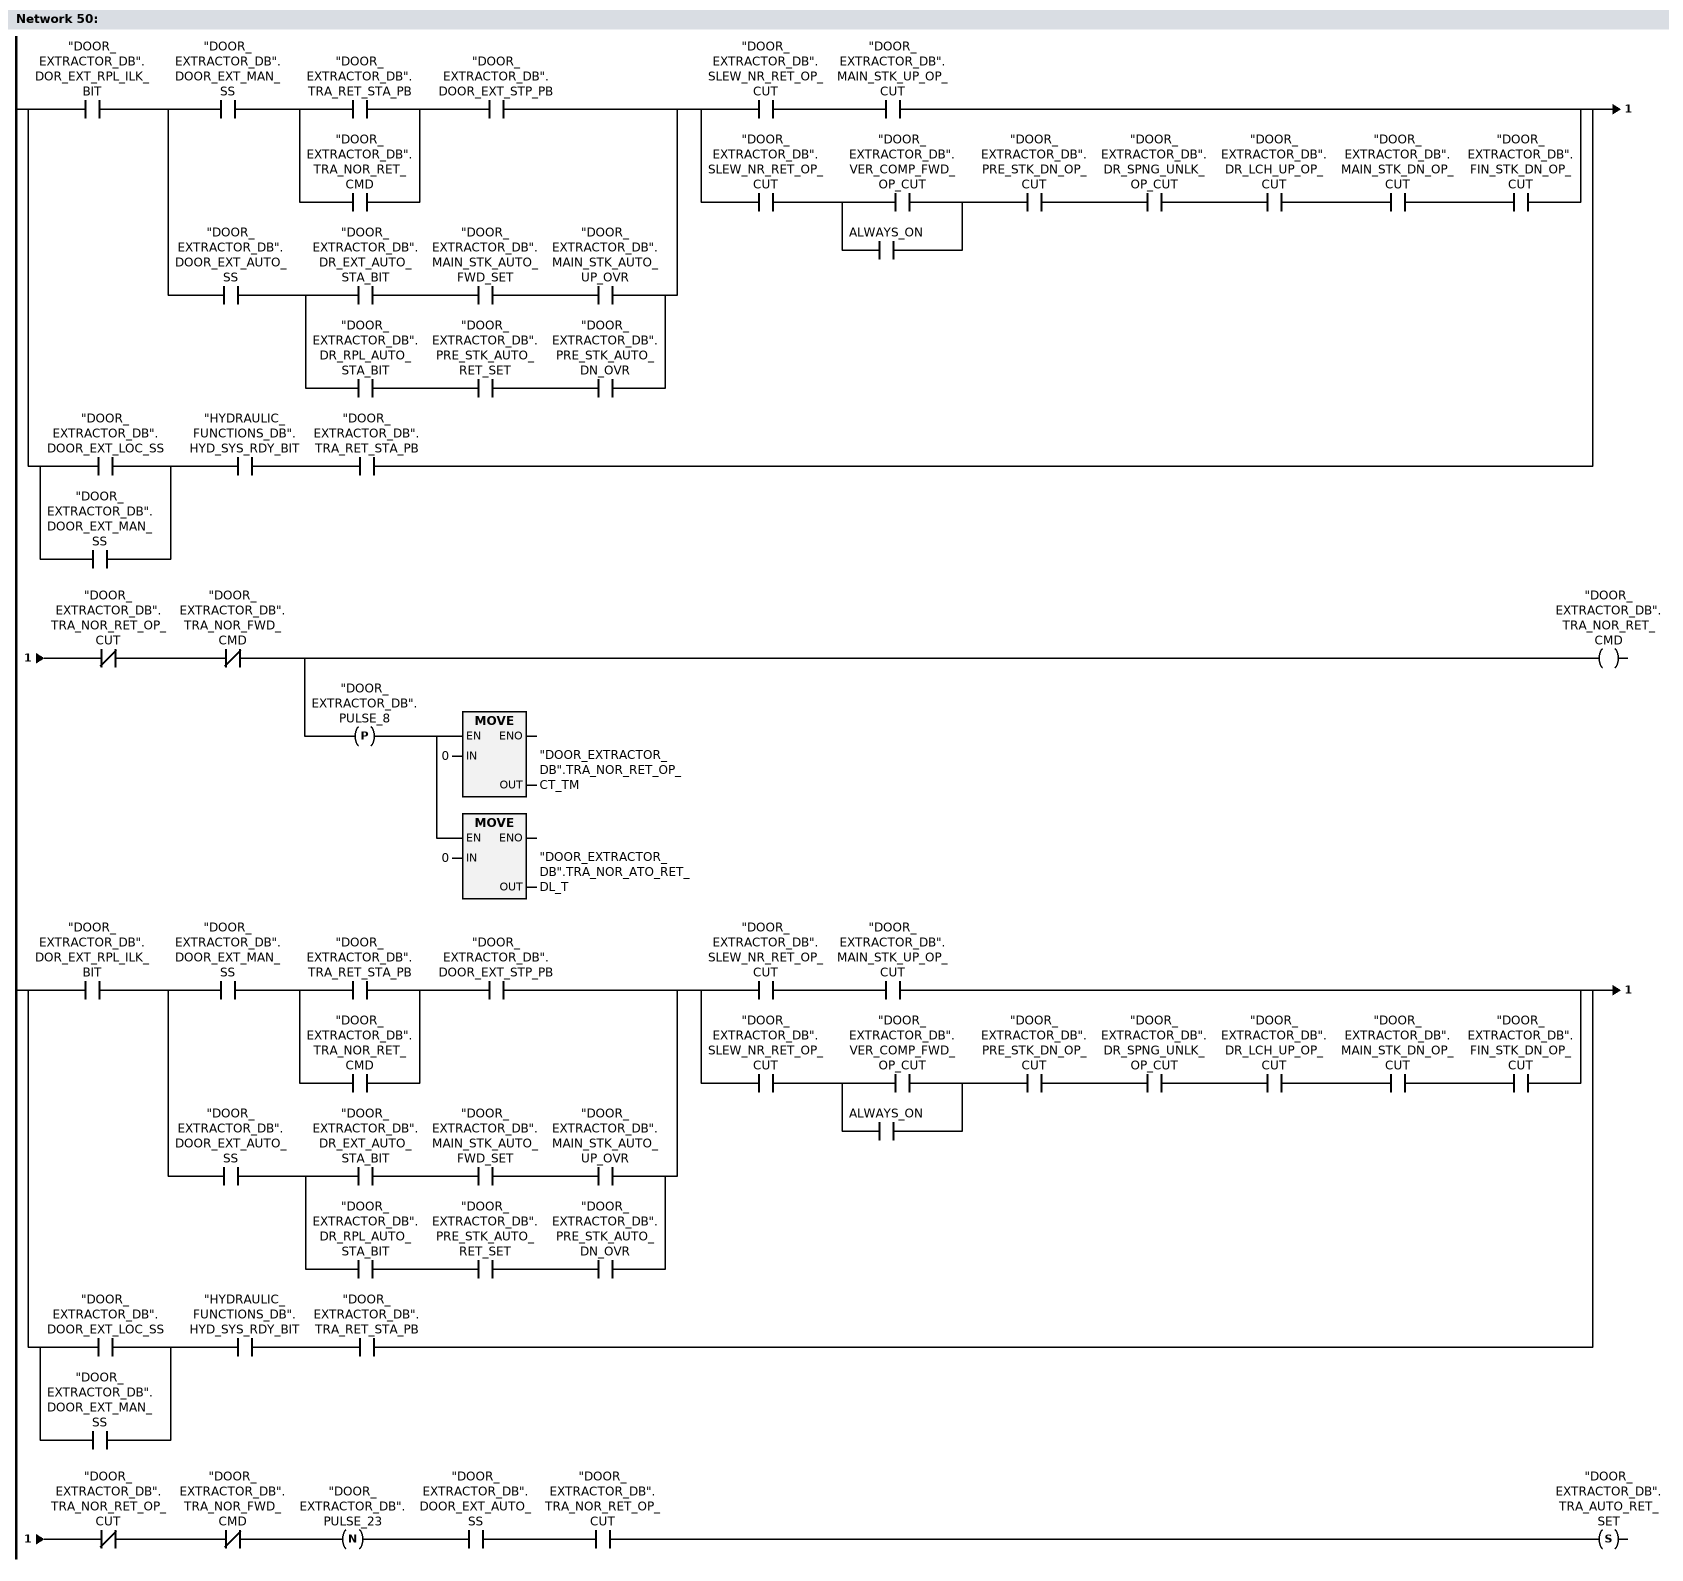
NETWORK
TITLE =
      A(;
      A     "DOOR_EXTRACTOR_DB".DOR_EXT_RPL_ILK_BIT;
      A(;
      A     "DOOR_EXTRACTOR_DB".DOOR_EXT_MAN_SS;
      A(;
      O     "DOOR_EXTRACTOR_DB".TRA_RET_STA_PB;
      O     "DOOR_EXTRACTOR_DB".TRA_NOR_RET_CMD;
      );
      A     "DOOR_EXTRACTOR_DB".DOOR_EXT_STP_PB;
      O;
      A     "DOOR_EXTRACTOR_DB".DOOR_EXT_AUTO_SS;
      A(;
      A     "DOOR_EXTRACTOR_DB".DR_EXT_AUTO_STA_BIT;
      A     "DOOR_EXTRACTOR_DB".MAIN_STK_AUTO_FWD_SET;
      A     "DOOR_EXTRACTOR_DB".MAIN_STK_AUTO_UP_OVR;
      O;
      A     "DOOR_EXTRACTOR_DB".DR_RPL_AUTO_STA_BIT;
      A     "DOOR_EXTRACTOR_DB".PRE_STK_AUTO_RET_SET;
      A     "DOOR_EXTRACTOR_DB".PRE_STK_AUTO_DN_OVR;
      );
      );
      A(;
      A     "DOOR_EXTRACTOR_DB".SLEW_NR_RET_OP_CUT;
      A     "DOOR_EXTRACTOR_DB".MAIN_STK_UP_OP_CUT;
      O;
      A     "DOOR_EXTRACTOR_DB".SLEW_NR_RET_OP_CUT;
      A(;
      O     "DOOR_EXTRACTOR_DB".VER_COMP_FWD_OP_CUT;
      O     "ALWAYS_ON";
      );
      A     "DOOR_EXTRACTOR_DB".PRE_STK_DN_OP_CUT;
      A     "DOOR_EXTRACTOR_DB".DR_SPNG_UNLK_OP_CUT;
      A     "DOOR_EXTRACTOR_DB".DR_LCH_UP_OP_CUT;
      A     "DOOR_EXTRACTOR_DB".MAIN_STK_DN_OP_CUT;
      A     "DOOR_EXTRACTOR_DB".FIN_STK_DN_OP_CUT;
      );
      O;
      A(;
      O     "DOOR_EXTRACTOR_DB".DOOR_EXT_LOC_SS;
      O     "DOOR_EXTRACTOR_DB".DOOR_EXT_MAN_SS;
      );
      A     "HYDRAULIC_FUNCTIONS_DB".HYD_SYS_RDY_BIT;
      A     "DOOR_EXTRACTOR_DB".TRA_RET_STA_PB;
      );
      AN    "DOOR_EXTRACTOR_DB".TRA_NOR_RET_OP_CUT;
      AN    "DOOR_EXTRACTOR_DB".TRA_NOR_FWD_CMD;
      =     L 0.0;
      A     L 0.0;
      BLD   102;
      =     "DOOR_EXTRACTOR_DB".TRA_NOR_RET_CMD;
      A(;
      A     L 0.0;
      FN    "DOOR_EXTRACTOR_DB".PULSE_23;
      );
      A     "DOOR_EXTRACTOR_DB".DOOR_EXT_AUTO_SS;
      A     "DOOR_EXTRACTOR_DB".TRA_NOR_RET_OP_CUT;
      S     "DOOR_EXTRACTOR_DB".TRA_AUTO_RET_SET;
      A     L 0.0;
      FP    "DOOR_EXTRACTOR_DB".PULSE_8;
      =     L 0.1;
      A     L 0.1;
      JNB   _02b;
      L     0;
      T     "DOOR_EXTRACTOR_DB".TRA_NOR_RET_OP_CT_TM;
_02b: NOP   0;
      A     L 0.1;
      JNB   _02c;
      L     0;
      T     "DOOR_EXTRACTOR_DB".TRA_NOR_ATO_RET_DL_T;
_02c: NOP   0;
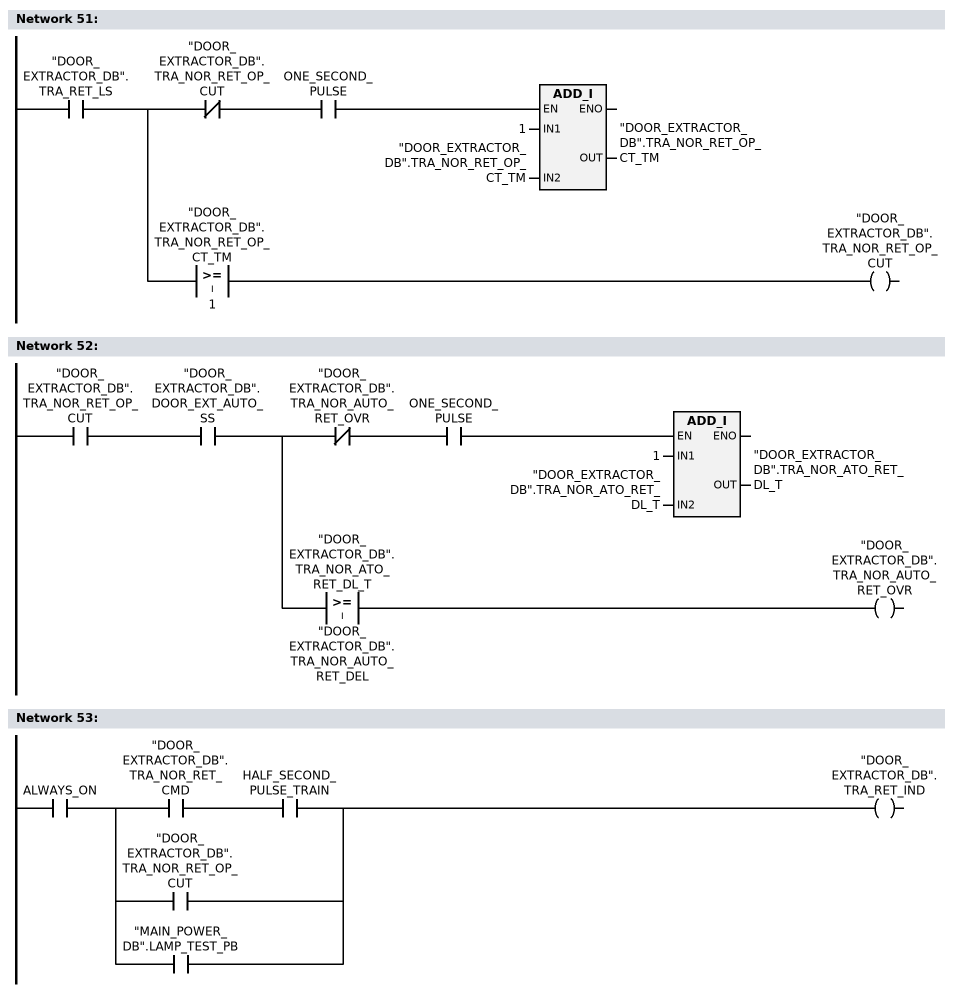
NETWORK
TITLE =
      A     "DOOR_EXTRACTOR_DB".TRA_RET_LS;
      =     L 0.0;
      A     L 0.0;
      AN    "DOOR_EXTRACTOR_DB".TRA_NOR_RET_OP_CUT;
      A     "ONE_SECOND_PULSE";
      JNB   _02d;
      L     1;
      L     "DOOR_EXTRACTOR_DB".TRA_NOR_RET_OP_CT_TM;
      +I;
      T     "DOOR_EXTRACTOR_DB".TRA_NOR_RET_OP_CT_TM;
_02d: NOP   0;
      A     L 0.0;
      A(;
      L     "DOOR_EXTRACTOR_DB".TRA_NOR_RET_OP_CT_TM;
      L     1;
      >=I;
      );
      =     "DOOR_EXTRACTOR_DB".TRA_NOR_RET_OP_CUT;
NETWORK
TITLE =
      A     "DOOR_EXTRACTOR_DB".TRA_NOR_RET_OP_CUT;
      A     "DOOR_EXTRACTOR_DB".DOOR_EXT_AUTO_SS;
      =     L 0.0;
      A     L 0.0;
      AN    "DOOR_EXTRACTOR_DB".TRA_NOR_AUTO_RET_OVR;
      A     "ONE_SECOND_PULSE";
      JNB   _02e;
      L     1;
      L     "DOOR_EXTRACTOR_DB".TRA_NOR_ATO_RET_DL_T;
      +I;
      T     "DOOR_EXTRACTOR_DB".TRA_NOR_ATO_RET_DL_T;
_02e: NOP   0;
      A     L 0.0;
      A(;
      L     "DOOR_EXTRACTOR_DB".TRA_NOR_ATO_RET_DL_T;
      L     "DOOR_EXTRACTOR_DB".TRA_NOR_AUTO_RET_DEL;
      >=I;
      );
      =     "DOOR_EXTRACTOR_DB".TRA_NOR_AUTO_RET_OVR;
NETWORK
TITLE =
      A     "ALWAYS_ON";
      A(;
      A     "DOOR_EXTRACTOR_DB".TRA_NOR_RET_CMD;
      A     "HALF_SECOND_PULSE_TRAIN";
      O     "DOOR_EXTRACTOR_DB".TRA_NOR_RET_OP_CUT;
      O     "MAIN_POWER_DB".LAMP_TEST_PB;
      );
      =     "DOOR_EXTRACTOR_DB".TRA_RET_IND;
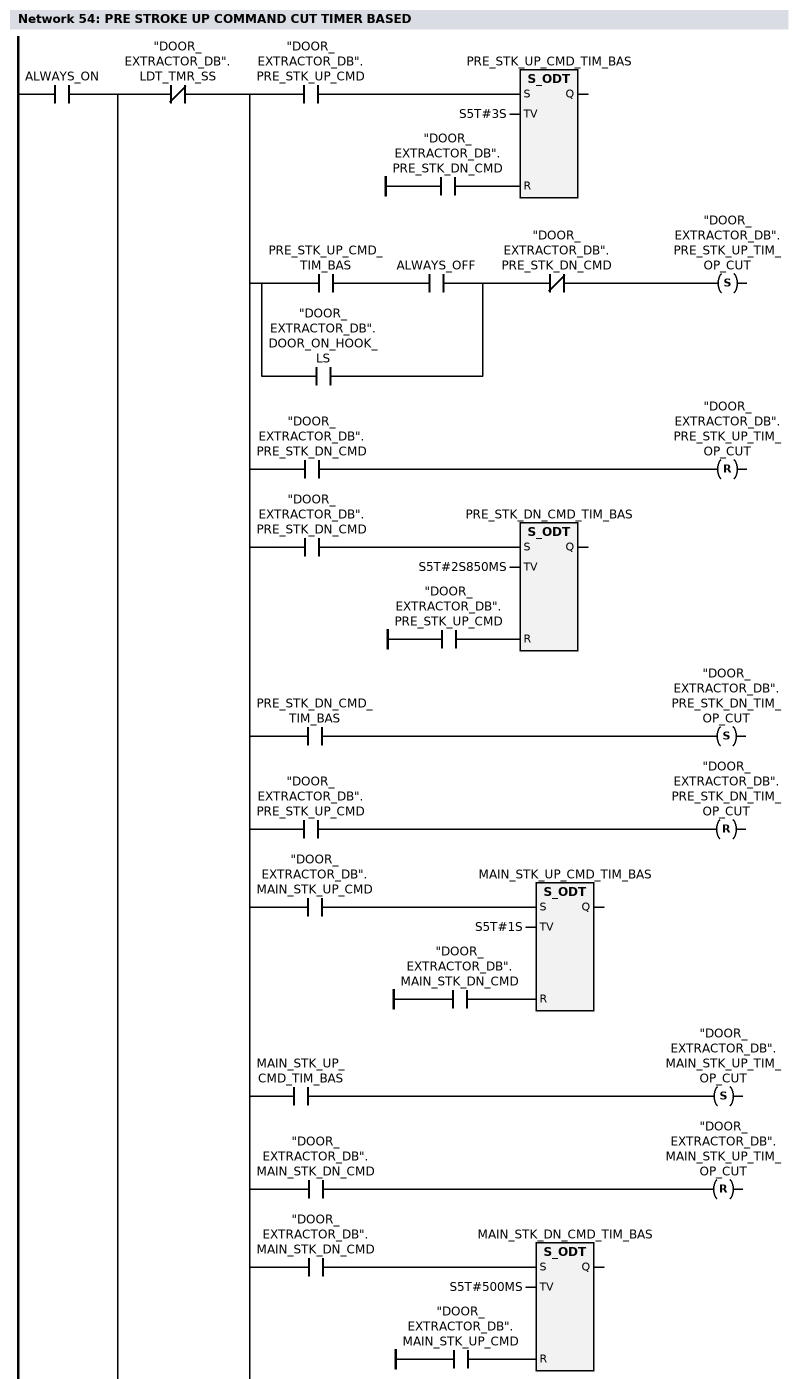
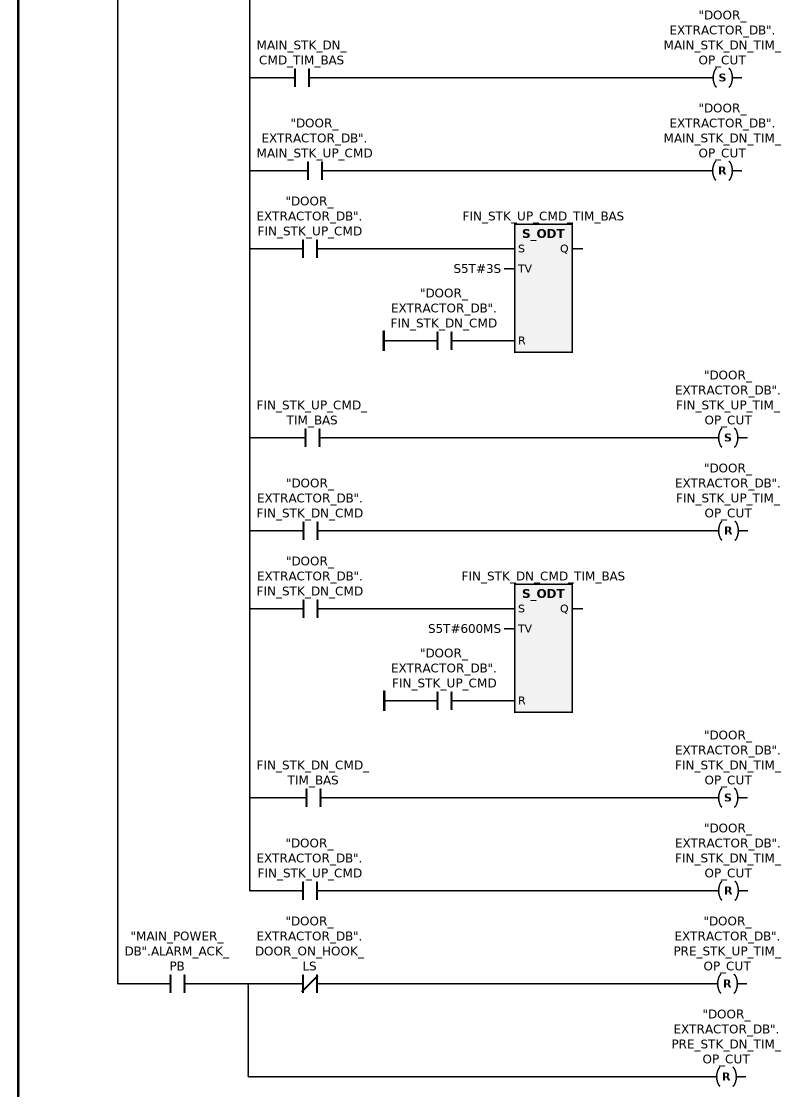
NETWORK
TITLE = PRE STROKE UP COMMAND CUT TIMER BASED
      A     "ALWAYS_ON";
      =     L 0.0;
      A     L 0.0;
      AN    "DOOR_EXTRACTOR_DB".LDT_TMR_SS;
      =     L 0.1;
      A     L 0.1;
      A     "DOOR_EXTRACTOR_DB".PRE_STK_UP_CMD;
      L     S5T#3S;
      SD    "PRE_STK_UP_CMD_TIM_BAS";
      A     "DOOR_EXTRACTOR_DB".PRE_STK_DN_CMD;
      R     "PRE_STK_UP_CMD_TIM_BAS";
      NOP   0;
      NOP   0;
      NOP   0;
      A     L 0.1;
      A(;
      A     "PRE_STK_UP_CMD_TIM_BAS";
      A     "ALWAYS_OFF";
      O     "DOOR_EXTRACTOR_DB".DOOR_ON_HOOK_LS;
      );
      AN    "DOOR_EXTRACTOR_DB".PRE_STK_DN_CMD;
      S     "DOOR_EXTRACTOR_DB".PRE_STK_UP_TIM_OP_CUT;
      A     L 0.1;
      A     "DOOR_EXTRACTOR_DB".PRE_STK_DN_CMD;
      R     "DOOR_EXTRACTOR_DB".PRE_STK_UP_TIM_OP_CUT;
      A     L 0.1;
      A     "DOOR_EXTRACTOR_DB".PRE_STK_DN_CMD;
      L     S5T#2S850MS;
      SD    "PRE_STK_DN_CMD_TIM_BAS";
      A     "DOOR_EXTRACTOR_DB".PRE_STK_UP_CMD;
      R     "PRE_STK_DN_CMD_TIM_BAS";
      NOP   0;
      NOP   0;
      NOP   0;
      A     L 0.1;
      A     "PRE_STK_DN_CMD_TIM_BAS";
      S     "DOOR_EXTRACTOR_DB".PRE_STK_DN_TIM_OP_CUT;
      A     L 0.1;
      A     "DOOR_EXTRACTOR_DB".PRE_STK_UP_CMD;
      R     "DOOR_EXTRACTOR_DB".PRE_STK_DN_TIM_OP_CUT;
      A     L 0.1;
      A     "DOOR_EXTRACTOR_DB".MAIN_STK_UP_CMD;
      L     S5T#1S;
      SD    "MAIN_STK_UP_CMD_TIM_BAS";
      A     "DOOR_EXTRACTOR_DB".MAIN_STK_DN_CMD;
      R     "MAIN_STK_UP_CMD_TIM_BAS";
      NOP   0;
      NOP   0;
      NOP   0;
      A     L 0.1;
      A     "MAIN_STK_UP_CMD_TIM_BAS";
      S     "DOOR_EXTRACTOR_DB".MAIN_STK_UP_TIM_OP_CUT;
      A     L 0.1;
      A     "DOOR_EXTRACTOR_DB".MAIN_STK_DN_CMD;
      R     "DOOR_EXTRACTOR_DB".MAIN_STK_UP_TIM_OP_CUT;
      A     L 0.1;
      A     "DOOR_EXTRACTOR_DB".MAIN_STK_DN_CMD;
      L     S5T#500MS;
      SD    "MAIN_STK_DN_CMD_TIM_BAS";
      A     "DOOR_EXTRACTOR_DB".MAIN_STK_UP_CMD;
      R     "MAIN_STK_DN_CMD_TIM_BAS";
      NOP   0;
      NOP   0;
      NOP   0;
      A     L 0.1;
      A     "MAIN_STK_DN_CMD_TIM_BAS";
      S     "DOOR_EXTRACTOR_DB".MAIN_STK_DN_TIM_OP_CUT;
      A     L 0.1;
      A     "DOOR_EXTRACTOR_DB".MAIN_STK_UP_CMD;
      R     "DOOR_EXTRACTOR_DB".MAIN_STK_DN_TIM_OP_CUT;
      A     L 0.1;
      A     "DOOR_EXTRACTOR_DB".FIN_STK_UP_CMD;
      L     S5T#3S;
      SD    "FIN_STK_UP_CMD_TIM_BAS";
      A     "DOOR_EXTRACTOR_DB".FIN_STK_DN_CMD;
      R     "FIN_STK_UP_CMD_TIM_BAS";
      NOP   0;
      NOP   0;
      NOP   0;
      A     L 0.1;
      A     "FIN_STK_UP_CMD_TIM_BAS";
      S     "DOOR_EXTRACTOR_DB".FIN_STK_UP_TIM_OP_CUT;
      A     L 0.1;
      A     "DOOR_EXTRACTOR_DB".FIN_STK_DN_CMD;
      R     "DOOR_EXTRACTOR_DB".FIN_STK_UP_TIM_OP_CUT;
      A     L 0.1;
      A     "DOOR_EXTRACTOR_DB".FIN_STK_DN_CMD;
      L     S5T#600MS;
      SD    "FIN_STK_DN_CMD_TIM_BAS";
      A     "DOOR_EXTRACTOR_DB".FIN_STK_UP_CMD;
      R     "FIN_STK_DN_CMD_TIM_BAS";
      NOP   0;
      NOP   0;
      NOP   0;
      A     L 0.1;
      A     "FIN_STK_DN_CMD_TIM_BAS";
      S     "DOOR_EXTRACTOR_DB".FIN_STK_DN_TIM_OP_CUT;
      A     L 0.1;
      A     "DOOR_EXTRACTOR_DB".FIN_STK_UP_CMD;
      R     "DOOR_EXTRACTOR_DB".FIN_STK_DN_TIM_OP_CUT;
      A     L 0.0;
      A     "MAIN_POWER_DB".ALARM_ACK_PB;
      =     L 0.1;
      A     L 0.1;
      AN    "DOOR_EXTRACTOR_DB".DOOR_ON_HOOK_LS;
      R     "DOOR_EXTRACTOR_DB".PRE_STK_UP_TIM_OP_CUT;
      A     L 0.1;
      BLD   102;
      R     "DOOR_EXTRACTOR_DB".PRE_STK_DN_TIM_OP_CUT;
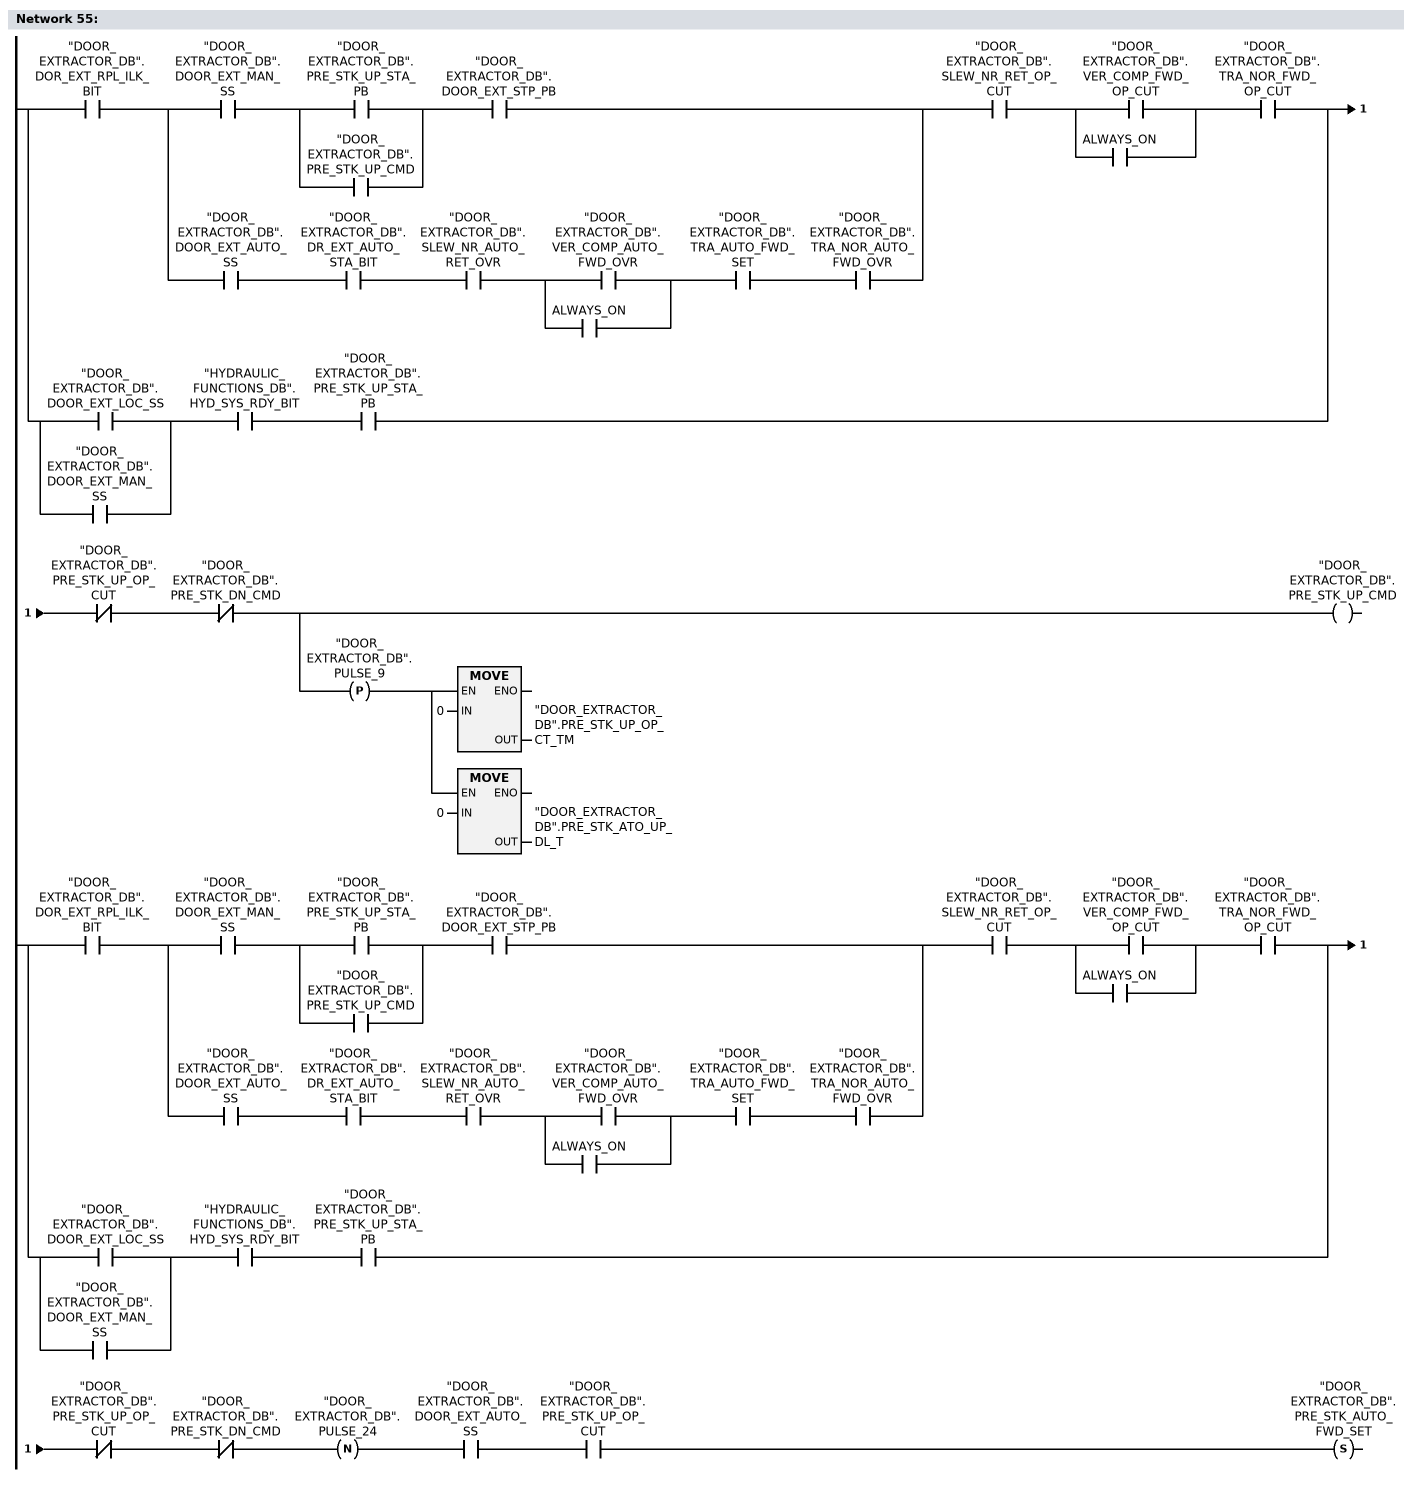
NETWORK
TITLE =
      A(;
      A     "DOOR_EXTRACTOR_DB".DOR_EXT_RPL_ILK_BIT;
      A(;
      A     "DOOR_EXTRACTOR_DB".DOOR_EXT_MAN_SS;
      A(;
      O     "DOOR_EXTRACTOR_DB".PRE_STK_UP_STA_PB;
      O     "DOOR_EXTRACTOR_DB".PRE_STK_UP_CMD;
      );
      A     "DOOR_EXTRACTOR_DB".DOOR_EXT_STP_PB;
      O;
      A     "DOOR_EXTRACTOR_DB".DOOR_EXT_AUTO_SS;
      A     "DOOR_EXTRACTOR_DB".DR_EXT_AUTO_STA_BIT;
      A     "DOOR_EXTRACTOR_DB".SLEW_NR_AUTO_RET_OVR;
      A(;
      O     "DOOR_EXTRACTOR_DB".VER_COMP_AUTO_FWD_OVR;
      O     "ALWAYS_ON";
      );
      A     "DOOR_EXTRACTOR_DB".TRA_AUTO_FWD_SET;
      A     "DOOR_EXTRACTOR_DB".TRA_NOR_AUTO_FWD_OVR;
      );
      A     "DOOR_EXTRACTOR_DB".SLEW_NR_RET_OP_CUT;
      A(;
      O     "DOOR_EXTRACTOR_DB".VER_COMP_FWD_OP_CUT;
      O     "ALWAYS_ON";
      );
      A     "DOOR_EXTRACTOR_DB".TRA_NOR_FWD_OP_CUT;
      O;
      A(;
      O     "DOOR_EXTRACTOR_DB".DOOR_EXT_LOC_SS;
      O     "DOOR_EXTRACTOR_DB".DOOR_EXT_MAN_SS;
      );
      A     "HYDRAULIC_FUNCTIONS_DB".HYD_SYS_RDY_BIT;
      A     "DOOR_EXTRACTOR_DB".PRE_STK_UP_STA_PB;
      );
      AN    "DOOR_EXTRACTOR_DB".PRE_STK_UP_OP_CUT;
      AN    "DOOR_EXTRACTOR_DB".PRE_STK_DN_CMD;
      =     L 0.0;
      A     L 0.0;
      BLD   102;
      =     "DOOR_EXTRACTOR_DB".PRE_STK_UP_CMD;
      A(;
      A     L 0.0;
      FN    "DOOR_EXTRACTOR_DB".PULSE_24;
      );
      A     "DOOR_EXTRACTOR_DB".DOOR_EXT_AUTO_SS;
      A     "DOOR_EXTRACTOR_DB".PRE_STK_UP_OP_CUT;
      S     "DOOR_EXTRACTOR_DB".PRE_STK_AUTO_FWD_SET;
      A     L 0.0;
      FP    "DOOR_EXTRACTOR_DB".PULSE_9;
      =     L 0.1;
      A     L 0.1;
      JNB   _02f;
      L     0;
      T     "DOOR_EXTRACTOR_DB".PRE_STK_UP_OP_CT_TM;
_02f: NOP   0;
      A     L 0.1;
      JNB   _030;
      L     0;
      T     "DOOR_EXTRACTOR_DB".PRE_STK_ATO_UP_DL_T;
_030: NOP   0;
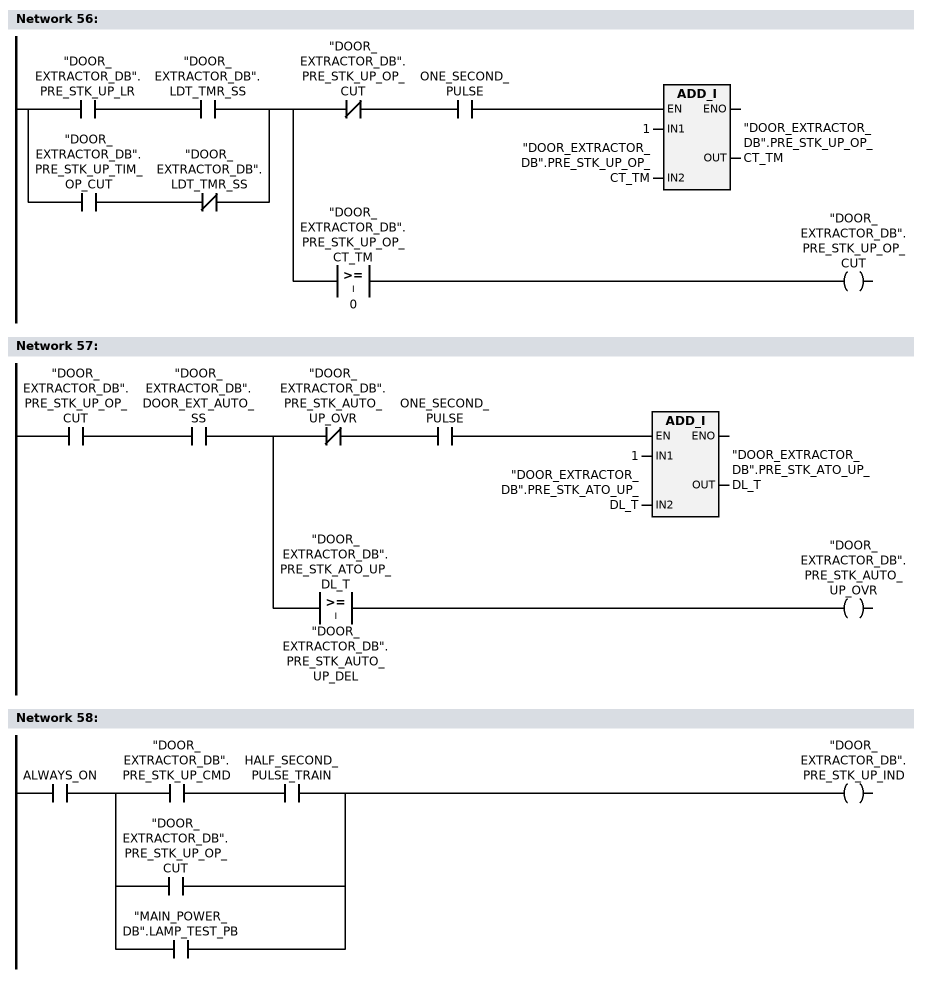
NETWORK
TITLE =
      A     "DOOR_EXTRACTOR_DB".PRE_STK_UP_LR;
      A     "DOOR_EXTRACTOR_DB".LDT_TMR_SS;
      O;
      A     "DOOR_EXTRACTOR_DB".PRE_STK_UP_TIM_OP_CUT;
      AN    "DOOR_EXTRACTOR_DB".LDT_TMR_SS;
      =     L 0.0;
      A     L 0.0;
      AN    "DOOR_EXTRACTOR_DB".PRE_STK_UP_OP_CUT;
      A     "ONE_SECOND_PULSE";
      JNB   _031;
      L     1;
      L     "DOOR_EXTRACTOR_DB".PRE_STK_UP_OP_CT_TM;
      +I;
      T     "DOOR_EXTRACTOR_DB".PRE_STK_UP_OP_CT_TM;
_031: NOP   0;
      A     L 0.0;
      A(;
      L     "DOOR_EXTRACTOR_DB".PRE_STK_UP_OP_CT_TM;
      L     0;
      >=I;
      );
      =     "DOOR_EXTRACTOR_DB".PRE_STK_UP_OP_CUT;
NETWORK
TITLE =
      A     "DOOR_EXTRACTOR_DB".PRE_STK_UP_OP_CUT;
      A     "DOOR_EXTRACTOR_DB".DOOR_EXT_AUTO_SS;
      =     L 0.0;
      A     L 0.0;
      AN    "DOOR_EXTRACTOR_DB".PRE_STK_AUTO_UP_OVR;
      A     "ONE_SECOND_PULSE";
      JNB   _032;
      L     1;
      L     "DOOR_EXTRACTOR_DB".PRE_STK_ATO_UP_DL_T;
      +I;
      T     "DOOR_EXTRACTOR_DB".PRE_STK_ATO_UP_DL_T;
_032: NOP   0;
      A     L 0.0;
      A(;
      L     "DOOR_EXTRACTOR_DB".PRE_STK_ATO_UP_DL_T;
      L     "DOOR_EXTRACTOR_DB".PRE_STK_AUTO_UP_DEL;
      >=I;
      );
      =     "DOOR_EXTRACTOR_DB".PRE_STK_AUTO_UP_OVR;
NETWORK
TITLE =
      A     "ALWAYS_ON";
      A(;
      A     "DOOR_EXTRACTOR_DB".PRE_STK_UP_CMD;
      A     "HALF_SECOND_PULSE_TRAIN";
      O     "DOOR_EXTRACTOR_DB".PRE_STK_UP_OP_CUT;
      O     "MAIN_POWER_DB".LAMP_TEST_PB;
      );
      =     "DOOR_EXTRACTOR_DB".PRE_STK_UP_IND;
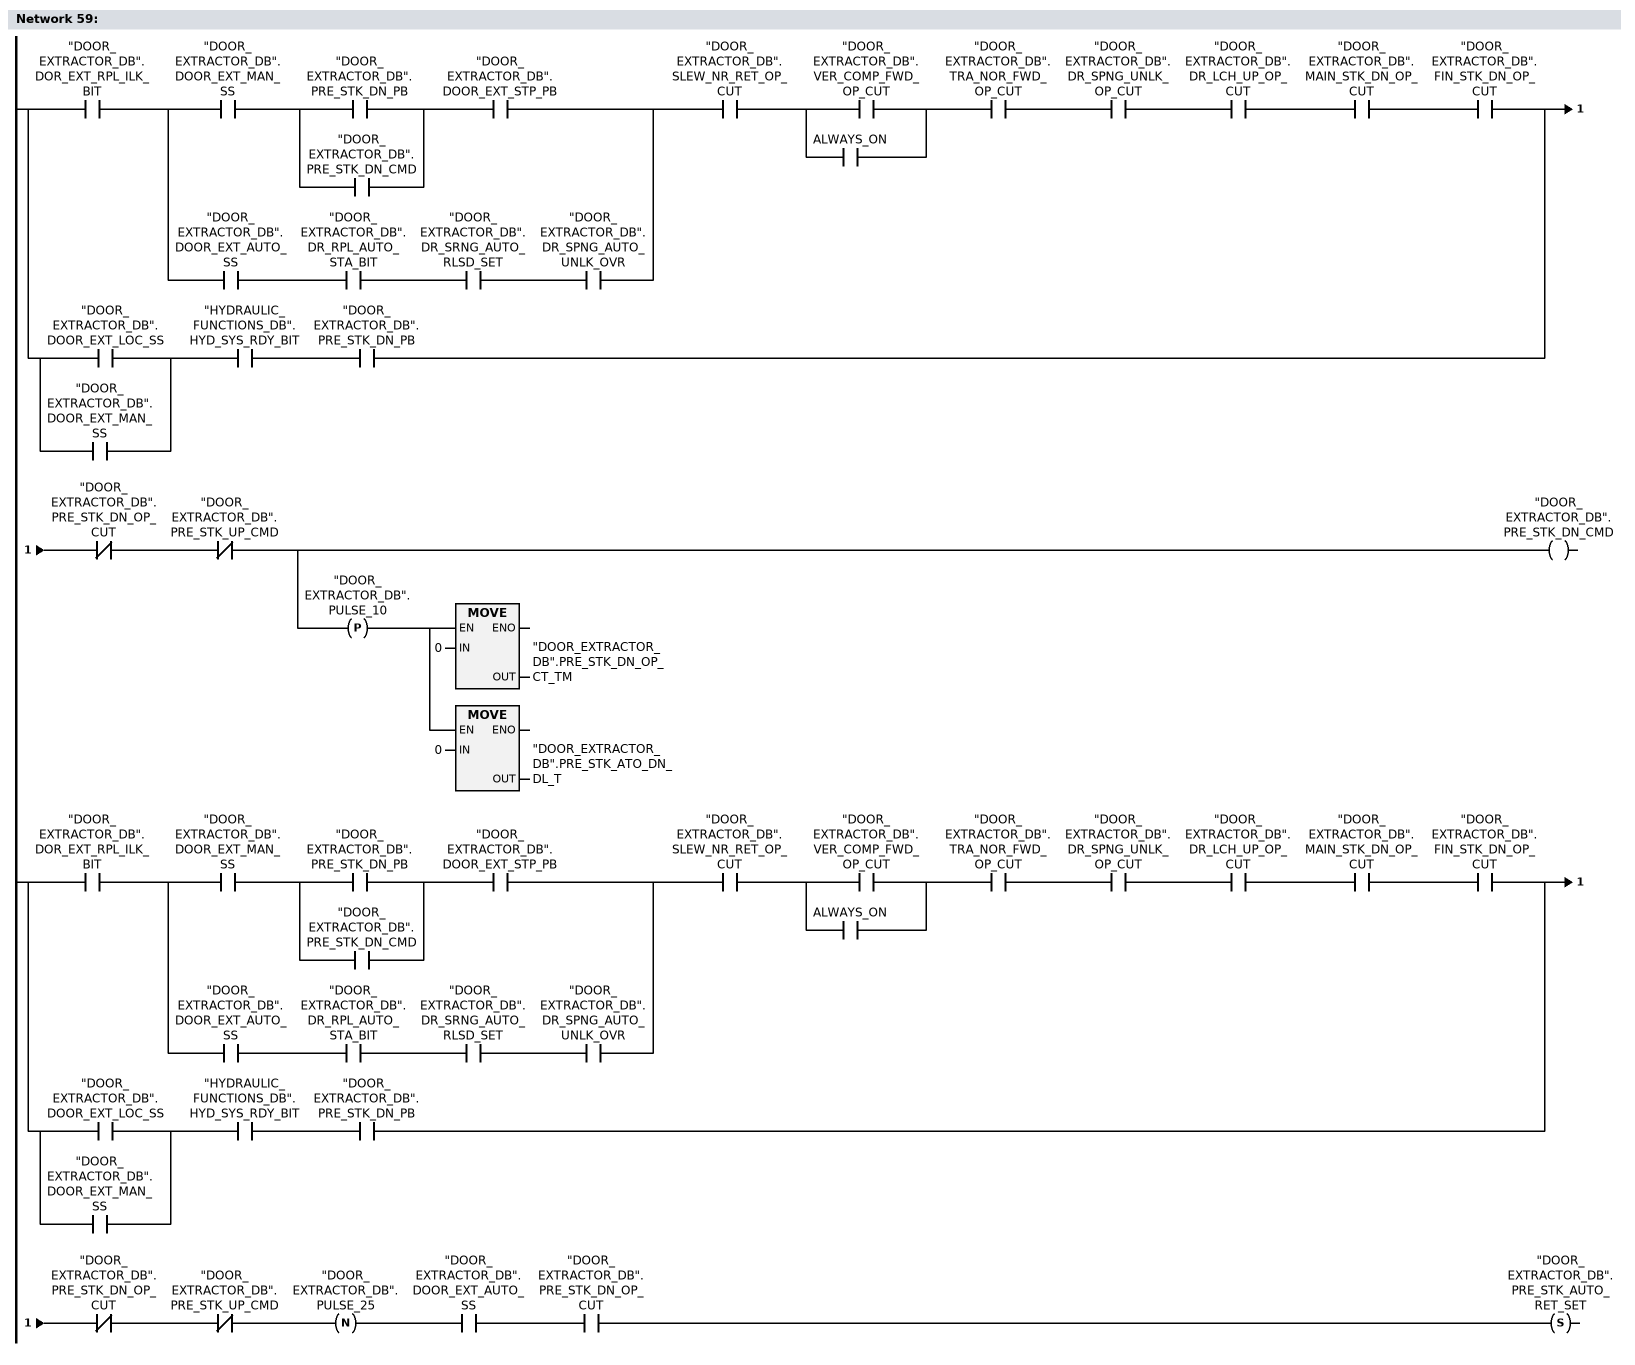
NETWORK
TITLE =
      A(;
      A     "DOOR_EXTRACTOR_DB".DOR_EXT_RPL_ILK_BIT;
      A(;
      A     "DOOR_EXTRACTOR_DB".DOOR_EXT_MAN_SS;
      A(;
      O     "DOOR_EXTRACTOR_DB".PRE_STK_DN_PB;
      O     "DOOR_EXTRACTOR_DB".PRE_STK_DN_CMD;
      );
      A     "DOOR_EXTRACTOR_DB".DOOR_EXT_STP_PB;
      O;
      A     "DOOR_EXTRACTOR_DB".DOOR_EXT_AUTO_SS;
      A     "DOOR_EXTRACTOR_DB".DR_RPL_AUTO_STA_BIT;
      A     "DOOR_EXTRACTOR_DB".DR_SRNG_AUTO_RLSD_SET;
      A     "DOOR_EXTRACTOR_DB".DR_SPNG_AUTO_UNLK_OVR;
      );
      A     "DOOR_EXTRACTOR_DB".SLEW_NR_RET_OP_CUT;
      A(;
      O     "DOOR_EXTRACTOR_DB".VER_COMP_FWD_OP_CUT;
      O     "ALWAYS_ON";
      );
      A     "DOOR_EXTRACTOR_DB".TRA_NOR_FWD_OP_CUT;
      A     "DOOR_EXTRACTOR_DB".DR_SPNG_UNLK_OP_CUT;
      A     "DOOR_EXTRACTOR_DB".DR_LCH_UP_OP_CUT;
      A     "DOOR_EXTRACTOR_DB".MAIN_STK_DN_OP_CUT;
      A     "DOOR_EXTRACTOR_DB".FIN_STK_DN_OP_CUT;
      O;
      A(;
      O     "DOOR_EXTRACTOR_DB".DOOR_EXT_LOC_SS;
      O     "DOOR_EXTRACTOR_DB".DOOR_EXT_MAN_SS;
      );
      A     "HYDRAULIC_FUNCTIONS_DB".HYD_SYS_RDY_BIT;
      A     "DOOR_EXTRACTOR_DB".PRE_STK_DN_PB;
      );
      AN    "DOOR_EXTRACTOR_DB".PRE_STK_DN_OP_CUT;
      AN    "DOOR_EXTRACTOR_DB".PRE_STK_UP_CMD;
      =     L 0.0;
      A     L 0.0;
      BLD   102;
      =     "DOOR_EXTRACTOR_DB".PRE_STK_DN_CMD;
      A(;
      A     L 0.0;
      FN    "DOOR_EXTRACTOR_DB".PULSE_25;
      );
      A     "DOOR_EXTRACTOR_DB".DOOR_EXT_AUTO_SS;
      A     "DOOR_EXTRACTOR_DB".PRE_STK_DN_OP_CUT;
      S     "DOOR_EXTRACTOR_DB".PRE_STK_AUTO_RET_SET;
      A     L 0.0;
      FP    "DOOR_EXTRACTOR_DB".PULSE_10;
      =     L 0.1;
      A     L 0.1;
      JNB   _033;
      L     0;
      T     "DOOR_EXTRACTOR_DB".PRE_STK_DN_OP_CT_TM;
_033: NOP   0;
      A     L 0.1;
      JNB   _034;
      L     0;
      T     "DOOR_EXTRACTOR_DB".PRE_STK_ATO_DN_DL_T;
_034: NOP   0;
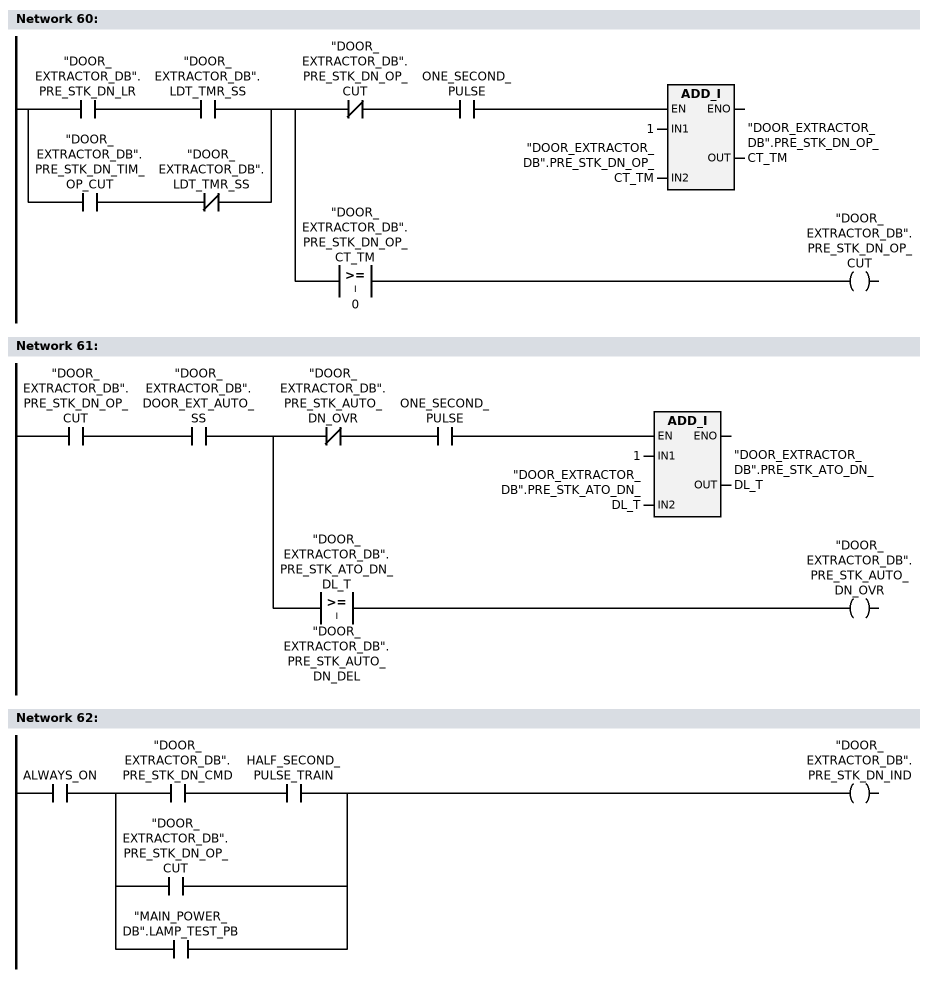
NETWORK
TITLE =
      A     "DOOR_EXTRACTOR_DB".PRE_STK_DN_LR;
      A     "DOOR_EXTRACTOR_DB".LDT_TMR_SS;
      O;
      A     "DOOR_EXTRACTOR_DB".PRE_STK_DN_TIM_OP_CUT;
      AN    "DOOR_EXTRACTOR_DB".LDT_TMR_SS;
      =     L 0.0;
      A     L 0.0;
      AN    "DOOR_EXTRACTOR_DB".PRE_STK_DN_OP_CUT;
      A     "ONE_SECOND_PULSE";
      JNB   _035;
      L     1;
      L     "DOOR_EXTRACTOR_DB".PRE_STK_DN_OP_CT_TM;
      +I;
      T     "DOOR_EXTRACTOR_DB".PRE_STK_DN_OP_CT_TM;
_035: NOP   0;
      A     L 0.0;
      A(;
      L     "DOOR_EXTRACTOR_DB".PRE_STK_DN_OP_CT_TM;
      L     0;
      >=I;
      );
      =     "DOOR_EXTRACTOR_DB".PRE_STK_DN_OP_CUT;
NETWORK
TITLE =
      A     "DOOR_EXTRACTOR_DB".PRE_STK_DN_OP_CUT;
      A     "DOOR_EXTRACTOR_DB".DOOR_EXT_AUTO_SS;
      =     L 0.0;
      A     L 0.0;
      AN    "DOOR_EXTRACTOR_DB".PRE_STK_AUTO_DN_OVR;
      A     "ONE_SECOND_PULSE";
      JNB   _036;
      L     1;
      L     "DOOR_EXTRACTOR_DB".PRE_STK_ATO_DN_DL_T;
      +I;
      T     "DOOR_EXTRACTOR_DB".PRE_STK_ATO_DN_DL_T;
_036: NOP   0;
      A     L 0.0;
      A(;
      L     "DOOR_EXTRACTOR_DB".PRE_STK_ATO_DN_DL_T;
      L     "DOOR_EXTRACTOR_DB".PRE_STK_AUTO_DN_DEL;
      >=I;
      );
      =     "DOOR_EXTRACTOR_DB".PRE_STK_AUTO_DN_OVR;
NETWORK
TITLE =
      A     "ALWAYS_ON";
      A(;
      A     "DOOR_EXTRACTOR_DB".PRE_STK_DN_CMD;
      A     "HALF_SECOND_PULSE_TRAIN";
      O     "DOOR_EXTRACTOR_DB".PRE_STK_DN_OP_CUT;
      O     "MAIN_POWER_DB".LAMP_TEST_PB;
      );
      =     "DOOR_EXTRACTOR_DB".PRE_STK_DN_IND;
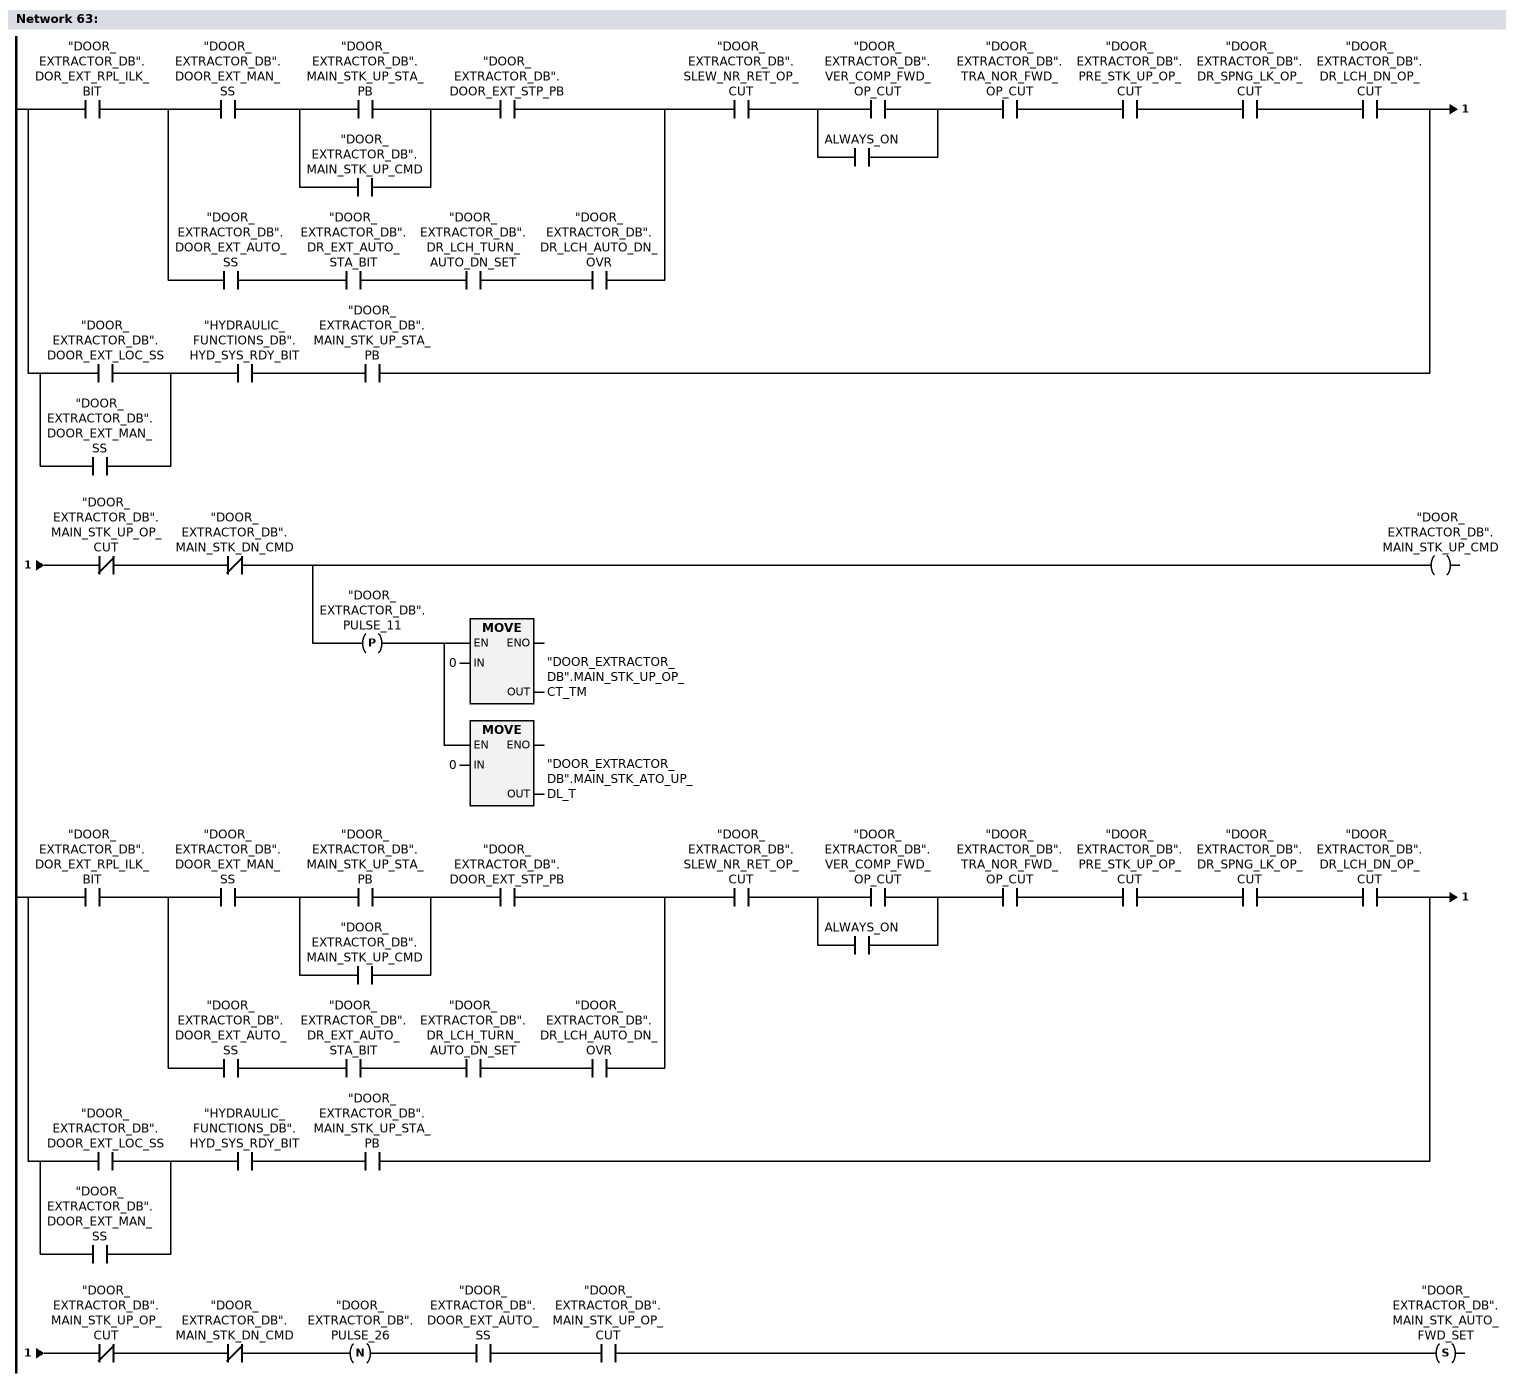
NETWORK
TITLE =
      A(;
      A     "DOOR_EXTRACTOR_DB".DOR_EXT_RPL_ILK_BIT;
      A(;
      A     "DOOR_EXTRACTOR_DB".DOOR_EXT_MAN_SS;
      A(;
      O     "DOOR_EXTRACTOR_DB".MAIN_STK_UP_STA_PB;
      O     "DOOR_EXTRACTOR_DB".MAIN_STK_UP_CMD;
      );
      A     "DOOR_EXTRACTOR_DB".DOOR_EXT_STP_PB;
      O;
      A     "DOOR_EXTRACTOR_DB".DOOR_EXT_AUTO_SS;
      A     "DOOR_EXTRACTOR_DB".DR_EXT_AUTO_STA_BIT;
      A     "DOOR_EXTRACTOR_DB".DR_LCH_TURN_AUTO_DN_SET;
      A     "DOOR_EXTRACTOR_DB".DR_LCH_AUTO_DN_OVR;
      );
      A     "DOOR_EXTRACTOR_DB".SLEW_NR_RET_OP_CUT;
      A(;
      O     "DOOR_EXTRACTOR_DB".VER_COMP_FWD_OP_CUT;
      O     "ALWAYS_ON";
      );
      A     "DOOR_EXTRACTOR_DB".TRA_NOR_FWD_OP_CUT;
      A     "DOOR_EXTRACTOR_DB".PRE_STK_UP_OP_CUT;
      A     "DOOR_EXTRACTOR_DB".DR_SPNG_LK_OP_CUT;
      A     "DOOR_EXTRACTOR_DB".DR_LCH_DN_OP_CUT;
      O;
      A(;
      O     "DOOR_EXTRACTOR_DB".DOOR_EXT_LOC_SS;
      O     "DOOR_EXTRACTOR_DB".DOOR_EXT_MAN_SS;
      );
      A     "HYDRAULIC_FUNCTIONS_DB".HYD_SYS_RDY_BIT;
      A     "DOOR_EXTRACTOR_DB".MAIN_STK_UP_STA_PB;
      );
      AN    "DOOR_EXTRACTOR_DB".MAIN_STK_UP_OP_CUT;
      AN    "DOOR_EXTRACTOR_DB".MAIN_STK_DN_CMD;
      =     L 0.0;
      A     L 0.0;
      BLD   102;
      =     "DOOR_EXTRACTOR_DB".MAIN_STK_UP_CMD;
      A(;
      A     L 0.0;
      FN    "DOOR_EXTRACTOR_DB".PULSE_26;
      );
      A     "DOOR_EXTRACTOR_DB".DOOR_EXT_AUTO_SS;
      A     "DOOR_EXTRACTOR_DB".MAIN_STK_UP_OP_CUT;
      S     "DOOR_EXTRACTOR_DB".MAIN_STK_AUTO_FWD_SET;
      A     L 0.0;
      FP    "DOOR_EXTRACTOR_DB".PULSE_11;
      =     L 0.1;
      A     L 0.1;
      JNB   _037;
      L     0;
      T     "DOOR_EXTRACTOR_DB".MAIN_STK_UP_OP_CT_TM;
_037: NOP   0;
      A     L 0.1;
      JNB   _038;
      L     0;
      T     "DOOR_EXTRACTOR_DB".MAIN_STK_ATO_UP_DL_T;
_038: NOP   0;
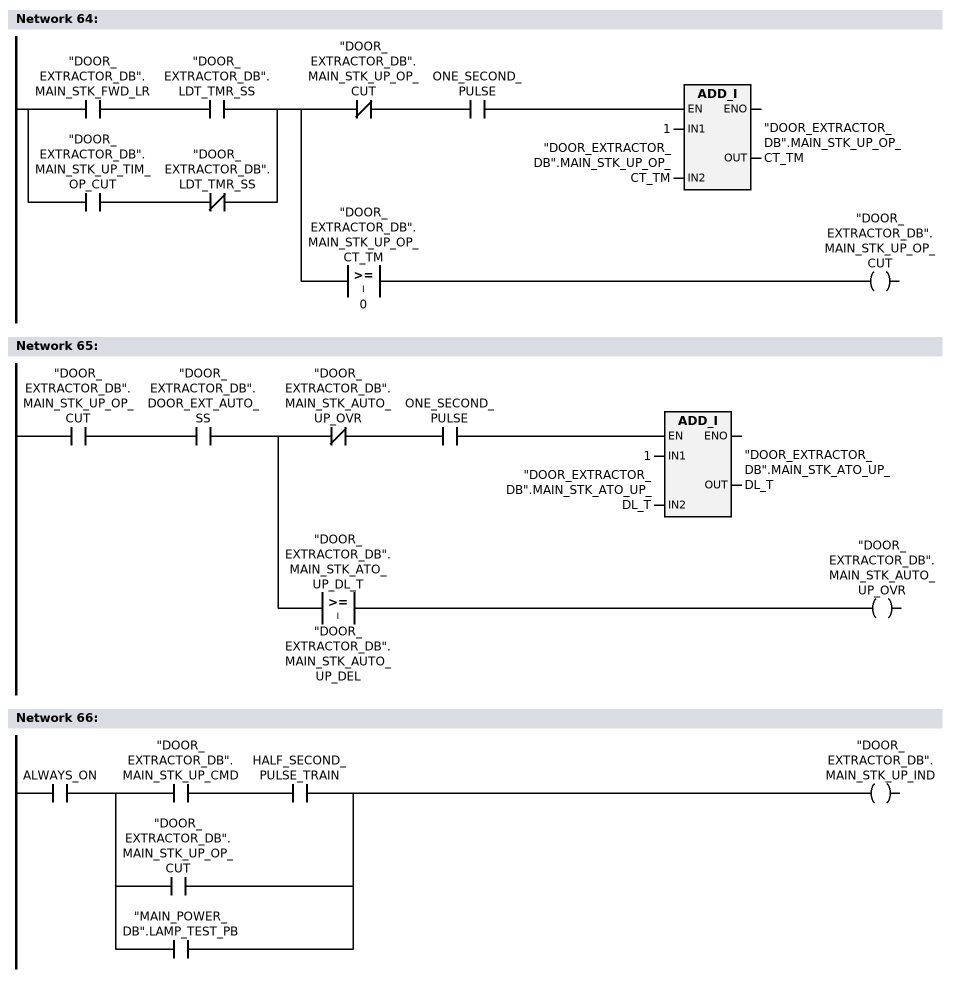
NETWORK
TITLE =
      A     "DOOR_EXTRACTOR_DB".MAIN_STK_FWD_LR;
      A     "DOOR_EXTRACTOR_DB".LDT_TMR_SS;
      O;
      A     "DOOR_EXTRACTOR_DB".MAIN_STK_UP_TIM_OP_CUT;
      AN    "DOOR_EXTRACTOR_DB".LDT_TMR_SS;
      =     L 0.0;
      A     L 0.0;
      AN    "DOOR_EXTRACTOR_DB".MAIN_STK_UP_OP_CUT;
      A     "ONE_SECOND_PULSE";
      JNB   _039;
      L     1;
      L     "DOOR_EXTRACTOR_DB".MAIN_STK_UP_OP_CT_TM;
      +I;
      T     "DOOR_EXTRACTOR_DB".MAIN_STK_UP_OP_CT_TM;
_039: NOP   0;
      A     L 0.0;
      A(;
      L     "DOOR_EXTRACTOR_DB".MAIN_STK_UP_OP_CT_TM;
      L     0;
      >=I;
      );
      =     "DOOR_EXTRACTOR_DB".MAIN_STK_UP_OP_CUT;
NETWORK
TITLE =
      A     "DOOR_EXTRACTOR_DB".MAIN_STK_UP_OP_CUT;
      A     "DOOR_EXTRACTOR_DB".DOOR_EXT_AUTO_SS;
      =     L 0.0;
      A     L 0.0;
      AN    "DOOR_EXTRACTOR_DB".MAIN_STK_AUTO_UP_OVR;
      A     "ONE_SECOND_PULSE";
      JNB   _03a;
      L     1;
      L     "DOOR_EXTRACTOR_DB".MAIN_STK_ATO_UP_DL_T;
      +I;
      T     "DOOR_EXTRACTOR_DB".MAIN_STK_ATO_UP_DL_T;
_03a: NOP   0;
      A     L 0.0;
      A(;
      L     "DOOR_EXTRACTOR_DB".MAIN_STK_ATO_UP_DL_T;
      L     "DOOR_EXTRACTOR_DB".MAIN_STK_AUTO_UP_DEL;
      >=I;
      );
      =     "DOOR_EXTRACTOR_DB".MAIN_STK_AUTO_UP_OVR;
NETWORK
TITLE =
      A     "ALWAYS_ON";
      A(;
      A     "DOOR_EXTRACTOR_DB".MAIN_STK_UP_CMD;
      A     "HALF_SECOND_PULSE_TRAIN";
      O     "DOOR_EXTRACTOR_DB".MAIN_STK_UP_OP_CUT;
      O     "MAIN_POWER_DB".LAMP_TEST_PB;
      );
      =     "DOOR_EXTRACTOR_DB".MAIN_STK_UP_IND;
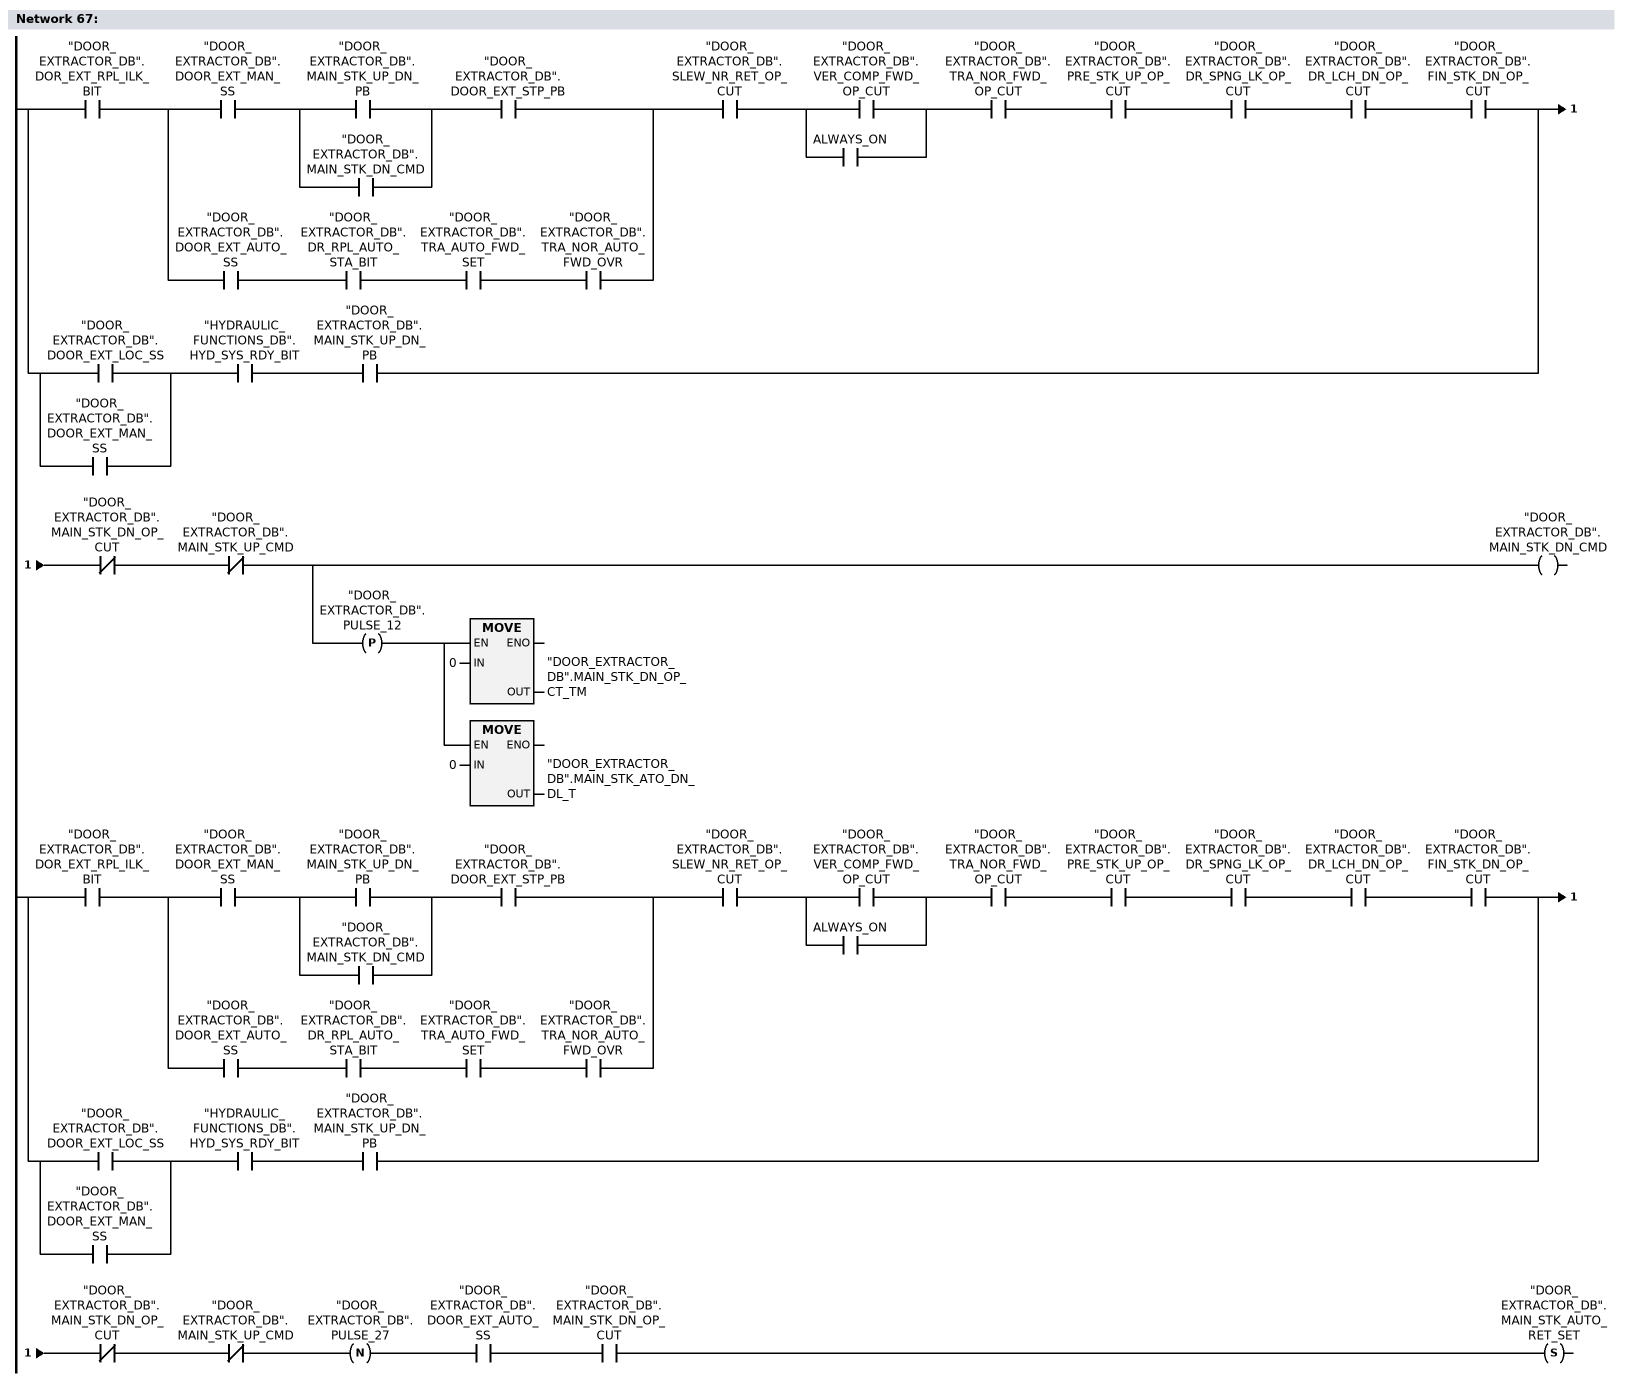
NETWORK
TITLE =
      A(;
      A     "DOOR_EXTRACTOR_DB".DOR_EXT_RPL_ILK_BIT;
      A(;
      A     "DOOR_EXTRACTOR_DB".DOOR_EXT_MAN_SS;
      A(;
      O     "DOOR_EXTRACTOR_DB".MAIN_STK_UP_DN_PB;
      O     "DOOR_EXTRACTOR_DB".MAIN_STK_DN_CMD;
      );
      A     "DOOR_EXTRACTOR_DB".DOOR_EXT_STP_PB;
      O;
      A     "DOOR_EXTRACTOR_DB".DOOR_EXT_AUTO_SS;
      A     "DOOR_EXTRACTOR_DB".DR_RPL_AUTO_STA_BIT;
      A     "DOOR_EXTRACTOR_DB".TRA_AUTO_FWD_SET;
      A     "DOOR_EXTRACTOR_DB".TRA_NOR_AUTO_FWD_OVR;
      );
      A     "DOOR_EXTRACTOR_DB".SLEW_NR_RET_OP_CUT;
      A(;
      O     "DOOR_EXTRACTOR_DB".VER_COMP_FWD_OP_CUT;
      O     "ALWAYS_ON";
      );
      A     "DOOR_EXTRACTOR_DB".TRA_NOR_FWD_OP_CUT;
      A     "DOOR_EXTRACTOR_DB".PRE_STK_UP_OP_CUT;
      A     "DOOR_EXTRACTOR_DB".DR_SPNG_LK_OP_CUT;
      A     "DOOR_EXTRACTOR_DB".DR_LCH_DN_OP_CUT;
      A     "DOOR_EXTRACTOR_DB".FIN_STK_DN_OP_CUT;
      O;
      A(;
      O     "DOOR_EXTRACTOR_DB".DOOR_EXT_LOC_SS;
      O     "DOOR_EXTRACTOR_DB".DOOR_EXT_MAN_SS;
      );
      A     "HYDRAULIC_FUNCTIONS_DB".HYD_SYS_RDY_BIT;
      A     "DOOR_EXTRACTOR_DB".MAIN_STK_UP_DN_PB;
      );
      AN    "DOOR_EXTRACTOR_DB".MAIN_STK_DN_OP_CUT;
      AN    "DOOR_EXTRACTOR_DB".MAIN_STK_UP_CMD;
      =     L 0.0;
      A     L 0.0;
      BLD   102;
      =     "DOOR_EXTRACTOR_DB".MAIN_STK_DN_CMD;
      A(;
      A     L 0.0;
      FN    "DOOR_EXTRACTOR_DB".PULSE_27;
      );
      A     "DOOR_EXTRACTOR_DB".DOOR_EXT_AUTO_SS;
      A     "DOOR_EXTRACTOR_DB".MAIN_STK_DN_OP_CUT;
      S     "DOOR_EXTRACTOR_DB".MAIN_STK_AUTO_RET_SET;
      A     L 0.0;
      FP    "DOOR_EXTRACTOR_DB".PULSE_12;
      =     L 0.1;
      A     L 0.1;
      JNB   _03b;
      L     0;
      T     "DOOR_EXTRACTOR_DB".MAIN_STK_DN_OP_CT_TM;
_03b: NOP   0;
      A     L 0.1;
      JNB   _03c;
      L     0;
      T     "DOOR_EXTRACTOR_DB".MAIN_STK_ATO_DN_DL_T;
_03c: NOP   0;
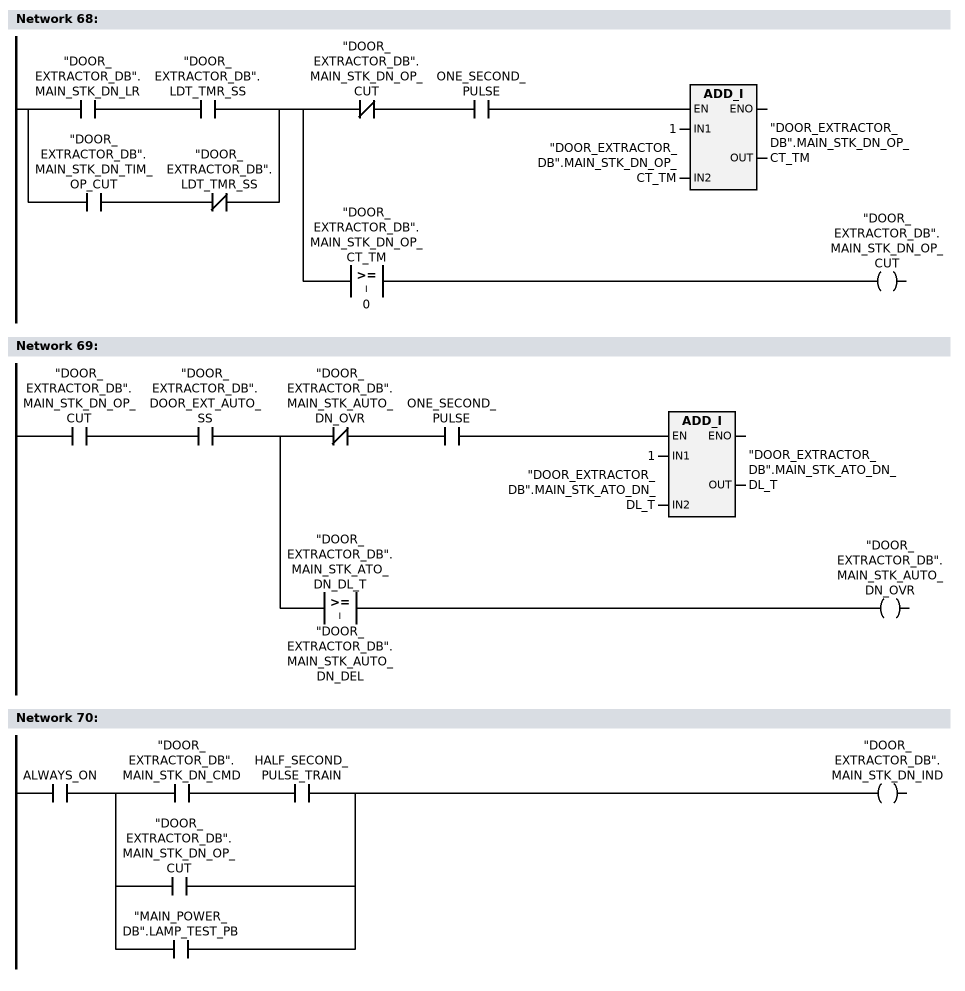
NETWORK
TITLE =
      A     "DOOR_EXTRACTOR_DB".MAIN_STK_DN_LR;
      A     "DOOR_EXTRACTOR_DB".LDT_TMR_SS;
      O;
      A     "DOOR_EXTRACTOR_DB".MAIN_STK_DN_TIM_OP_CUT;
      AN    "DOOR_EXTRACTOR_DB".LDT_TMR_SS;
      =     L 0.0;
      A     L 0.0;
      AN    "DOOR_EXTRACTOR_DB".MAIN_STK_DN_OP_CUT;
      A     "ONE_SECOND_PULSE";
      JNB   _03d;
      L     1;
      L     "DOOR_EXTRACTOR_DB".MAIN_STK_DN_OP_CT_TM;
      +I;
      T     "DOOR_EXTRACTOR_DB".MAIN_STK_DN_OP_CT_TM;
_03d: NOP   0;
      A     L 0.0;
      A(;
      L     "DOOR_EXTRACTOR_DB".MAIN_STK_DN_OP_CT_TM;
      L     0;
      >=I;
      );
      =     "DOOR_EXTRACTOR_DB".MAIN_STK_DN_OP_CUT;
NETWORK
TITLE =
      A     "DOOR_EXTRACTOR_DB".MAIN_STK_DN_OP_CUT;
      A     "DOOR_EXTRACTOR_DB".DOOR_EXT_AUTO_SS;
      =     L 0.0;
      A     L 0.0;
      AN    "DOOR_EXTRACTOR_DB".MAIN_STK_AUTO_DN_OVR;
      A     "ONE_SECOND_PULSE";
      JNB   _03e;
      L     1;
      L     "DOOR_EXTRACTOR_DB".MAIN_STK_ATO_DN_DL_T;
      +I;
      T     "DOOR_EXTRACTOR_DB".MAIN_STK_ATO_DN_DL_T;
_03e: NOP   0;
      A     L 0.0;
      A(;
      L     "DOOR_EXTRACTOR_DB".MAIN_STK_ATO_DN_DL_T;
      L     "DOOR_EXTRACTOR_DB".MAIN_STK_AUTO_DN_DEL;
      >=I;
      );
      =     "DOOR_EXTRACTOR_DB".MAIN_STK_AUTO_DN_OVR;
NETWORK
TITLE =
      A     "ALWAYS_ON";
      A(;
      A     "DOOR_EXTRACTOR_DB".MAIN_STK_DN_CMD;
      A     "HALF_SECOND_PULSE_TRAIN";
      O     "DOOR_EXTRACTOR_DB".MAIN_STK_DN_OP_CUT;
      O     "MAIN_POWER_DB".LAMP_TEST_PB;
      );
      =     "DOOR_EXTRACTOR_DB".MAIN_STK_DN_IND;
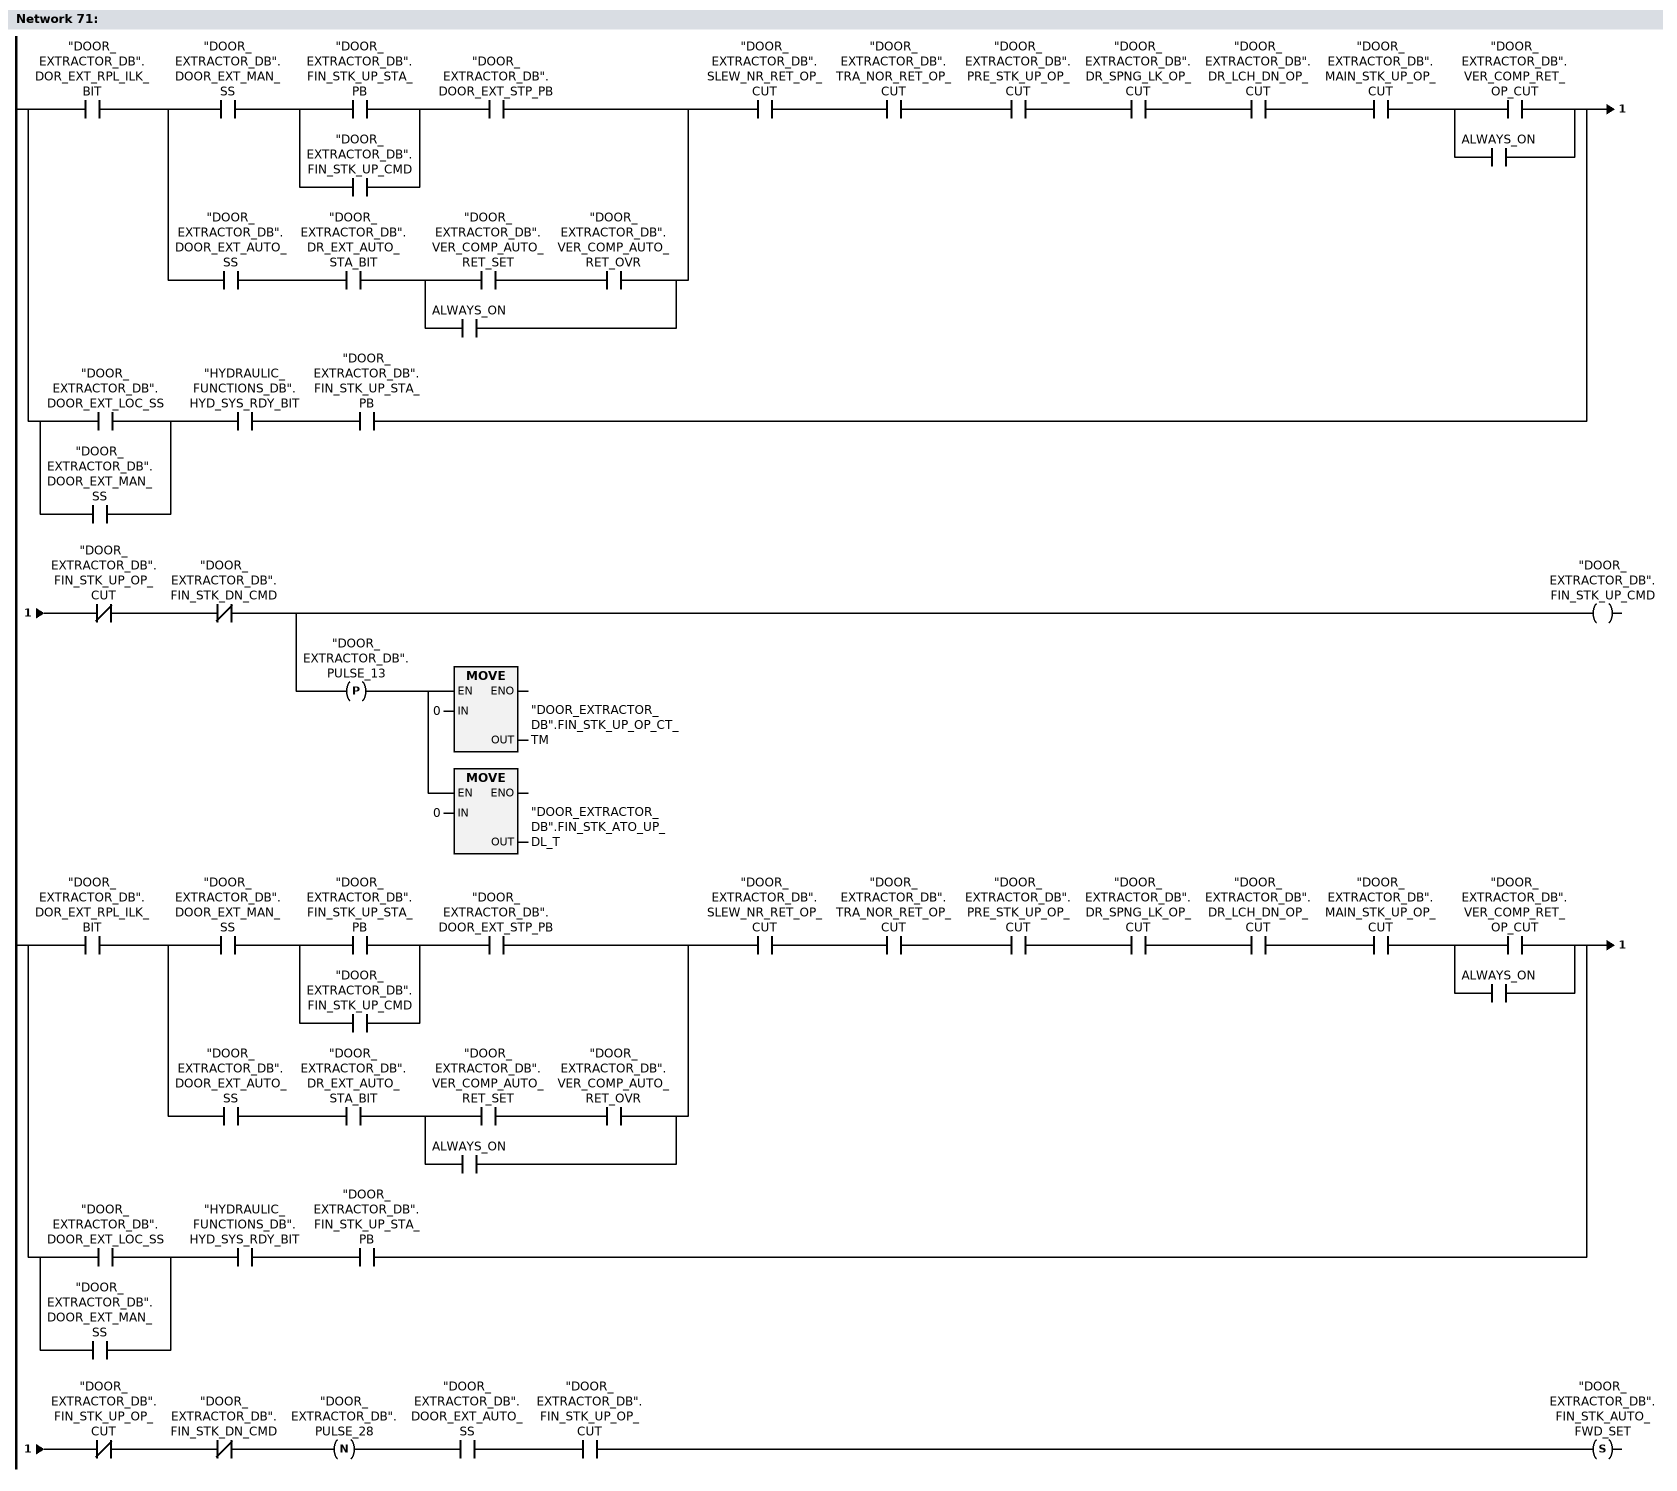
NETWORK
TITLE =
      A(;
      A     "DOOR_EXTRACTOR_DB".DOR_EXT_RPL_ILK_BIT;
      A(;
      A     "DOOR_EXTRACTOR_DB".DOOR_EXT_MAN_SS;
      A(;
      O     "DOOR_EXTRACTOR_DB".FIN_STK_UP_STA_PB;
      O     "DOOR_EXTRACTOR_DB".FIN_STK_UP_CMD;
      );
      A     "DOOR_EXTRACTOR_DB".DOOR_EXT_STP_PB;
      O;
      A     "DOOR_EXTRACTOR_DB".DOOR_EXT_AUTO_SS;
      A     "DOOR_EXTRACTOR_DB".DR_EXT_AUTO_STA_BIT;
      A(;
      A     "DOOR_EXTRACTOR_DB".VER_COMP_AUTO_RET_SET;
      A     "DOOR_EXTRACTOR_DB".VER_COMP_AUTO_RET_OVR;
      O     "ALWAYS_ON";
      );
      );
      A     "DOOR_EXTRACTOR_DB".SLEW_NR_RET_OP_CUT;
      A     "DOOR_EXTRACTOR_DB".TRA_NOR_RET_OP_CUT;
      A     "DOOR_EXTRACTOR_DB".PRE_STK_UP_OP_CUT;
      A     "DOOR_EXTRACTOR_DB".DR_SPNG_LK_OP_CUT;
      A     "DOOR_EXTRACTOR_DB".DR_LCH_DN_OP_CUT;
      A     "DOOR_EXTRACTOR_DB".MAIN_STK_UP_OP_CUT;
      A(;
      O     "DOOR_EXTRACTOR_DB".VER_COMP_RET_OP_CUT;
      O     "ALWAYS_ON";
      );
      O;
      A(;
      O     "DOOR_EXTRACTOR_DB".DOOR_EXT_LOC_SS;
      O     "DOOR_EXTRACTOR_DB".DOOR_EXT_MAN_SS;
      );
      A     "HYDRAULIC_FUNCTIONS_DB".HYD_SYS_RDY_BIT;
      A     "DOOR_EXTRACTOR_DB".FIN_STK_UP_STA_PB;
      );
      AN    "DOOR_EXTRACTOR_DB".FIN_STK_UP_OP_CUT;
      AN    "DOOR_EXTRACTOR_DB".FIN_STK_DN_CMD;
      =     L 0.0;
      A     L 0.0;
      BLD   102;
      =     "DOOR_EXTRACTOR_DB".FIN_STK_UP_CMD;
      A(;
      A     L 0.0;
      FN    "DOOR_EXTRACTOR_DB".PULSE_28;
      );
      A     "DOOR_EXTRACTOR_DB".DOOR_EXT_AUTO_SS;
      A     "DOOR_EXTRACTOR_DB".FIN_STK_UP_OP_CUT;
      S     "DOOR_EXTRACTOR_DB".FIN_STK_AUTO_FWD_SET;
      A     L 0.0;
      FP    "DOOR_EXTRACTOR_DB".PULSE_13;
      =     L 0.1;
      A     L 0.1;
      JNB   _03f;
      L     0;
      T     "DOOR_EXTRACTOR_DB".FIN_STK_UP_OP_CT_TM;
_03f: NOP   0;
      A     L 0.1;
      JNB   _040;
      L     0;
      T     "DOOR_EXTRACTOR_DB".FIN_STK_ATO_UP_DL_T;
_040: NOP   0;
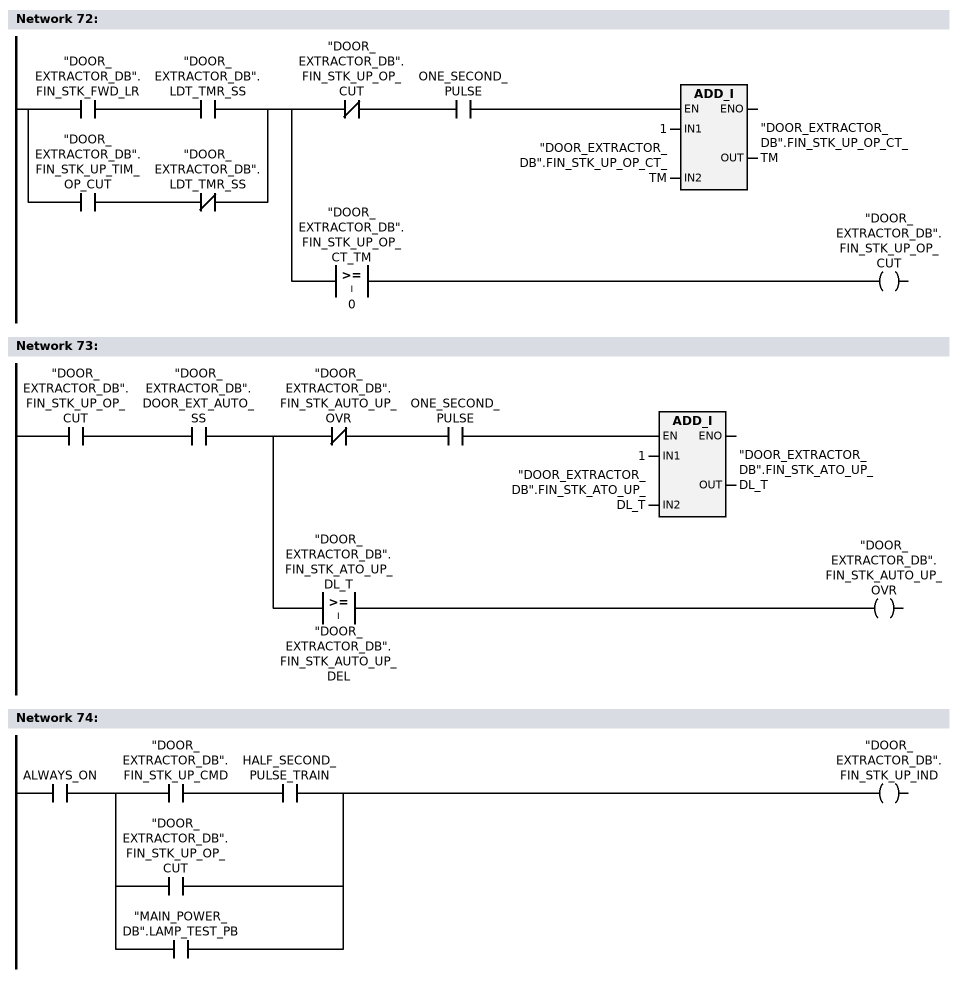
NETWORK
TITLE =
      A     "DOOR_EXTRACTOR_DB".FIN_STK_FWD_LR;
      A     "DOOR_EXTRACTOR_DB".LDT_TMR_SS;
      O;
      A     "DOOR_EXTRACTOR_DB".FIN_STK_UP_TIM_OP_CUT;
      AN    "DOOR_EXTRACTOR_DB".LDT_TMR_SS;
      =     L 0.0;
      A     L 0.0;
      AN    "DOOR_EXTRACTOR_DB".FIN_STK_UP_OP_CUT;
      A     "ONE_SECOND_PULSE";
      JNB   _041;
      L     1;
      L     "DOOR_EXTRACTOR_DB".FIN_STK_UP_OP_CT_TM;
      +I;
      T     "DOOR_EXTRACTOR_DB".FIN_STK_UP_OP_CT_TM;
_041: NOP   0;
      A     L 0.0;
      A(;
      L     "DOOR_EXTRACTOR_DB".FIN_STK_UP_OP_CT_TM;
      L     0;
      >=I;
      );
      =     "DOOR_EXTRACTOR_DB".FIN_STK_UP_OP_CUT;
NETWORK
TITLE =
      A     "DOOR_EXTRACTOR_DB".FIN_STK_UP_OP_CUT;
      A     "DOOR_EXTRACTOR_DB".DOOR_EXT_AUTO_SS;
      =     L 0.0;
      A     L 0.0;
      AN    "DOOR_EXTRACTOR_DB".FIN_STK_AUTO_UP_OVR;
      A     "ONE_SECOND_PULSE";
      JNB   _042;
      L     1;
      L     "DOOR_EXTRACTOR_DB".FIN_STK_ATO_UP_DL_T;
      +I;
      T     "DOOR_EXTRACTOR_DB".FIN_STK_ATO_UP_DL_T;
_042: NOP   0;
      A     L 0.0;
      A(;
      L     "DOOR_EXTRACTOR_DB".FIN_STK_ATO_UP_DL_T;
      L     "DOOR_EXTRACTOR_DB".FIN_STK_AUTO_UP_DEL;
      >=I;
      );
      =     "DOOR_EXTRACTOR_DB".FIN_STK_AUTO_UP_OVR;
NETWORK
TITLE =
      A     "ALWAYS_ON";
      A(;
      A     "DOOR_EXTRACTOR_DB".FIN_STK_UP_CMD;
      A     "HALF_SECOND_PULSE_TRAIN";
      O     "DOOR_EXTRACTOR_DB".FIN_STK_UP_OP_CUT;
      O     "MAIN_POWER_DB".LAMP_TEST_PB;
      );
      =     "DOOR_EXTRACTOR_DB".FIN_STK_UP_IND;
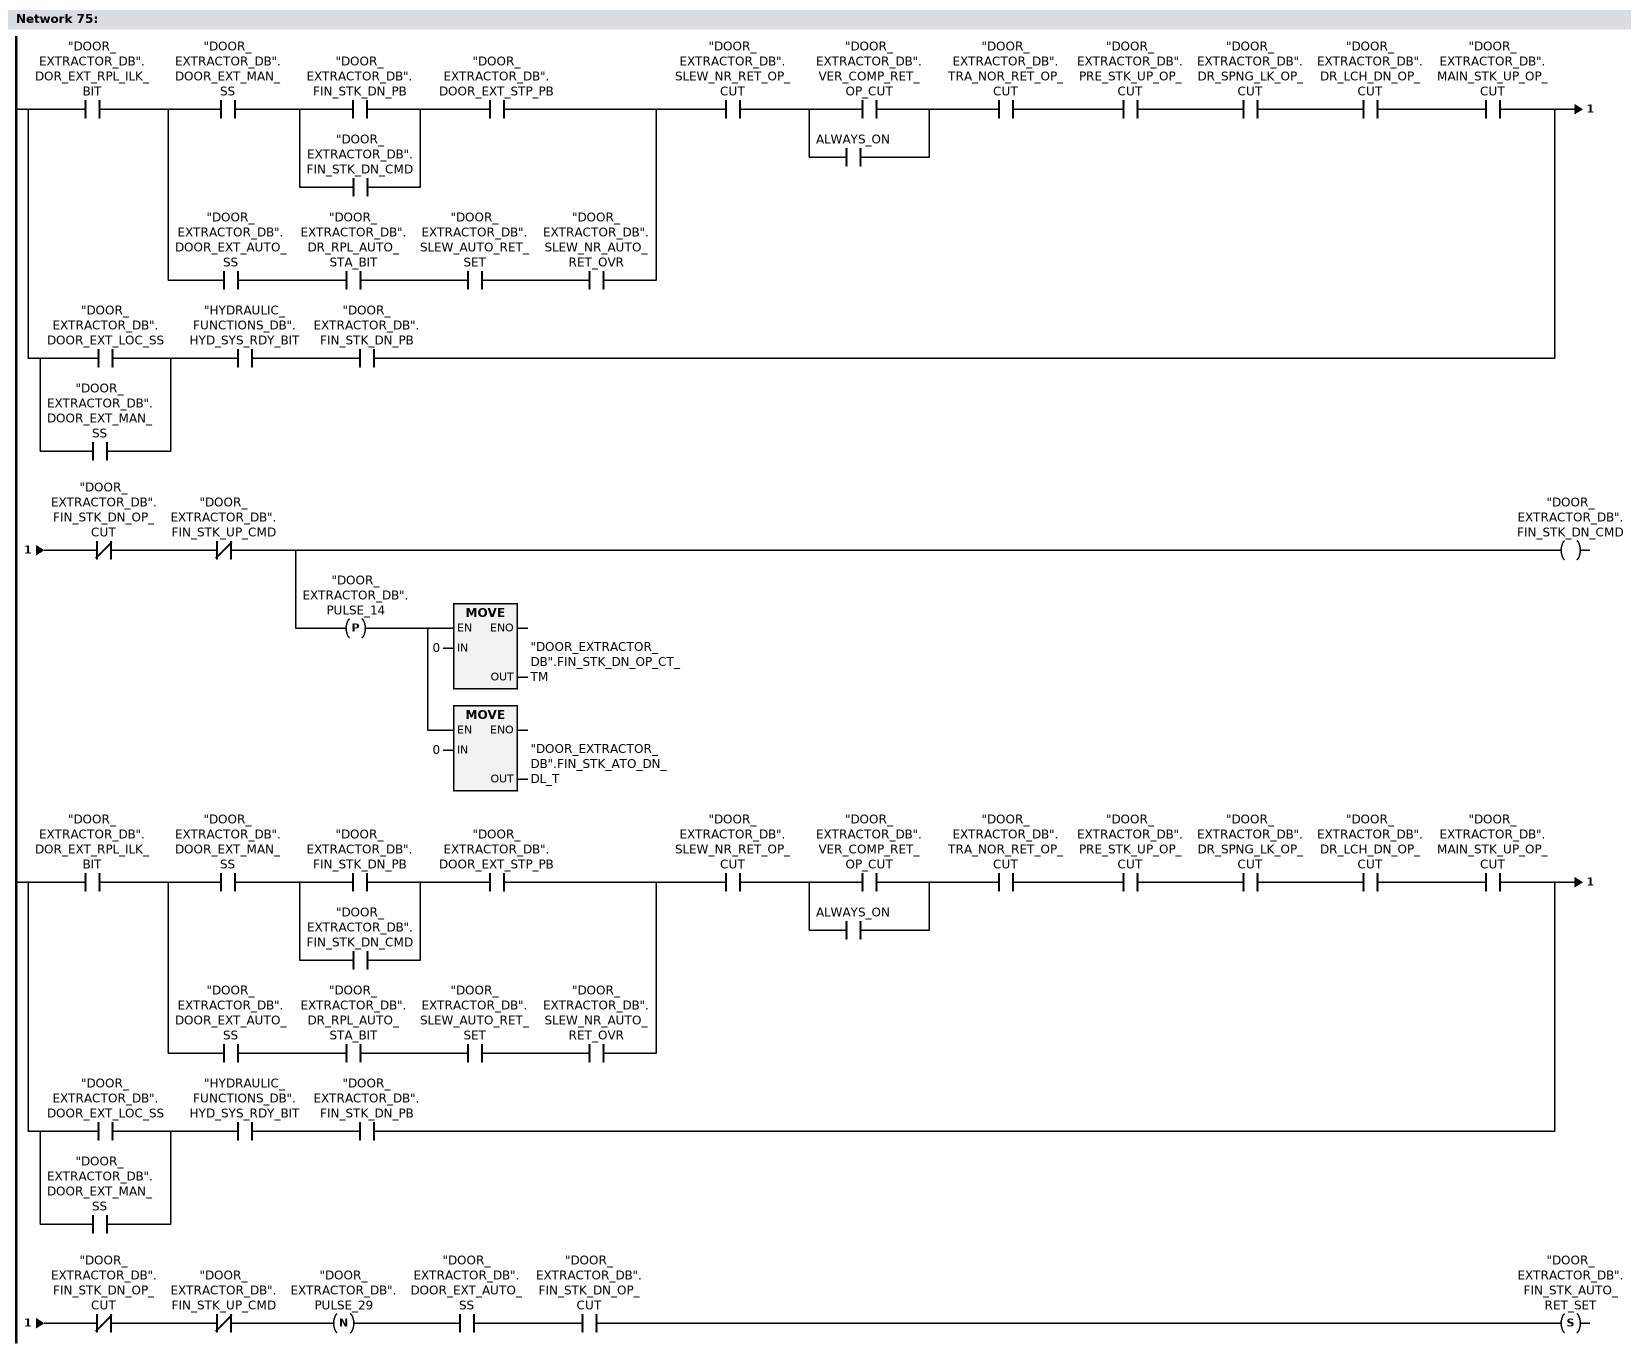
NETWORK
TITLE =
      A(;
      A     "DOOR_EXTRACTOR_DB".DOR_EXT_RPL_ILK_BIT;
      A(;
      A     "DOOR_EXTRACTOR_DB".DOOR_EXT_MAN_SS;
      A(;
      O     "DOOR_EXTRACTOR_DB".FIN_STK_DN_PB;
      O     "DOOR_EXTRACTOR_DB".FIN_STK_DN_CMD;
      );
      A     "DOOR_EXTRACTOR_DB".DOOR_EXT_STP_PB;
      O;
      A     "DOOR_EXTRACTOR_DB".DOOR_EXT_AUTO_SS;
      A     "DOOR_EXTRACTOR_DB".DR_RPL_AUTO_STA_BIT;
      A     "DOOR_EXTRACTOR_DB".SLEW_AUTO_RET_SET;
      A     "DOOR_EXTRACTOR_DB".SLEW_NR_AUTO_RET_OVR;
      );
      A     "DOOR_EXTRACTOR_DB".SLEW_NR_RET_OP_CUT;
      A(;
      O     "DOOR_EXTRACTOR_DB".VER_COMP_RET_OP_CUT;
      O     "ALWAYS_ON";
      );
      A     "DOOR_EXTRACTOR_DB".TRA_NOR_RET_OP_CUT;
      A     "DOOR_EXTRACTOR_DB".PRE_STK_UP_OP_CUT;
      A     "DOOR_EXTRACTOR_DB".DR_SPNG_LK_OP_CUT;
      A     "DOOR_EXTRACTOR_DB".DR_LCH_DN_OP_CUT;
      A     "DOOR_EXTRACTOR_DB".MAIN_STK_UP_OP_CUT;
      O;
      A(;
      O     "DOOR_EXTRACTOR_DB".DOOR_EXT_LOC_SS;
      O     "DOOR_EXTRACTOR_DB".DOOR_EXT_MAN_SS;
      );
      A     "HYDRAULIC_FUNCTIONS_DB".HYD_SYS_RDY_BIT;
      A     "DOOR_EXTRACTOR_DB".FIN_STK_DN_PB;
      );
      AN    "DOOR_EXTRACTOR_DB".FIN_STK_DN_OP_CUT;
      AN    "DOOR_EXTRACTOR_DB".FIN_STK_UP_CMD;
      =     L 0.0;
      A     L 0.0;
      BLD   102;
      =     "DOOR_EXTRACTOR_DB".FIN_STK_DN_CMD;
      A(;
      A     L 0.0;
      FN    "DOOR_EXTRACTOR_DB".PULSE_29;
      );
      A     "DOOR_EXTRACTOR_DB".DOOR_EXT_AUTO_SS;
      A     "DOOR_EXTRACTOR_DB".FIN_STK_DN_OP_CUT;
      S     "DOOR_EXTRACTOR_DB".FIN_STK_AUTO_RET_SET;
      A     L 0.0;
      FP    "DOOR_EXTRACTOR_DB".PULSE_14;
      =     L 0.1;
      A     L 0.1;
      JNB   _043;
      L     0;
      T     "DOOR_EXTRACTOR_DB".FIN_STK_DN_OP_CT_TM;
_043: NOP   0;
      A     L 0.1;
      JNB   _044;
      L     0;
      T     "DOOR_EXTRACTOR_DB".FIN_STK_ATO_DN_DL_T;
_044: NOP   0;
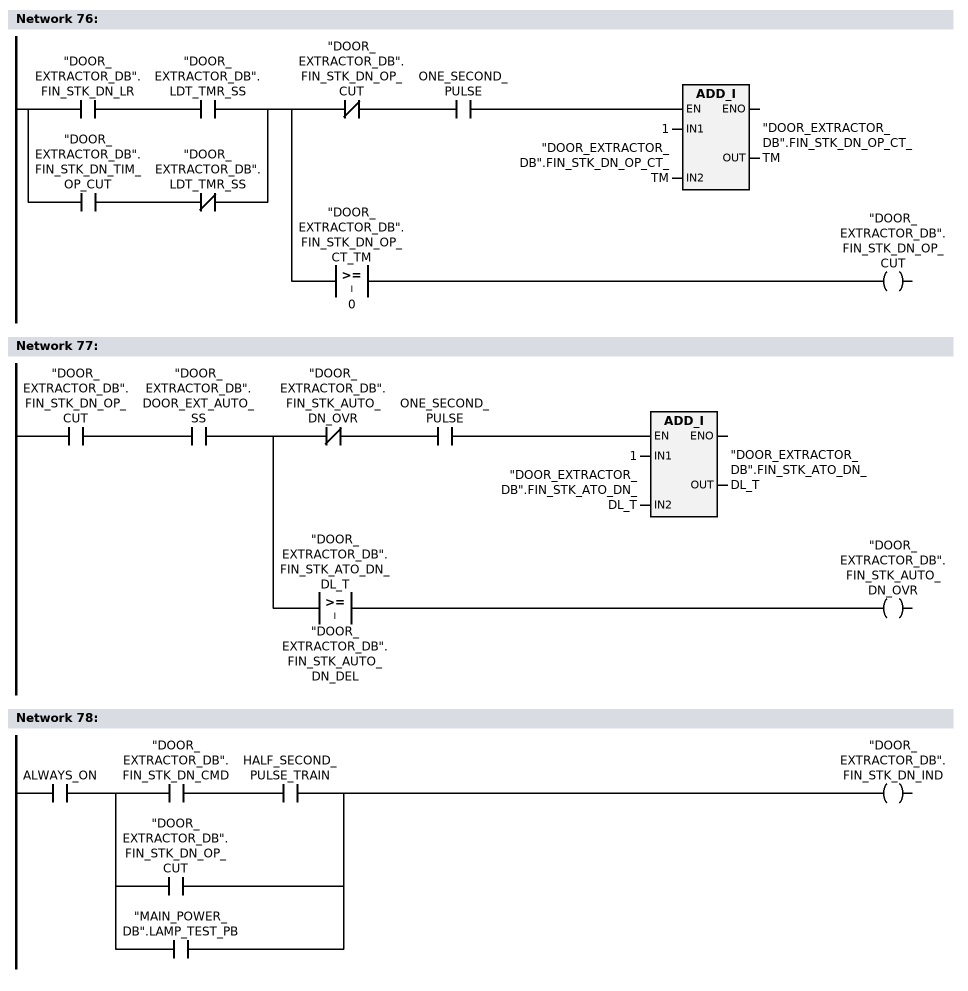
NETWORK
TITLE =
      A     "DOOR_EXTRACTOR_DB".FIN_STK_DN_LR;
      A     "DOOR_EXTRACTOR_DB".LDT_TMR_SS;
      O;
      A     "DOOR_EXTRACTOR_DB".FIN_STK_DN_TIM_OP_CUT;
      AN    "DOOR_EXTRACTOR_DB".LDT_TMR_SS;
      =     L 0.0;
      A     L 0.0;
      AN    "DOOR_EXTRACTOR_DB".FIN_STK_DN_OP_CUT;
      A     "ONE_SECOND_PULSE";
      JNB   _045;
      L     1;
      L     "DOOR_EXTRACTOR_DB".FIN_STK_DN_OP_CT_TM;
      +I;
      T     "DOOR_EXTRACTOR_DB".FIN_STK_DN_OP_CT_TM;
_045: NOP   0;
      A     L 0.0;
      A(;
      L     "DOOR_EXTRACTOR_DB".FIN_STK_DN_OP_CT_TM;
      L     0;
      >=I;
      );
      =     "DOOR_EXTRACTOR_DB".FIN_STK_DN_OP_CUT;
NETWORK
TITLE =
      A     "DOOR_EXTRACTOR_DB".FIN_STK_DN_OP_CUT;
      A     "DOOR_EXTRACTOR_DB".DOOR_EXT_AUTO_SS;
      =     L 0.0;
      A     L 0.0;
      AN    "DOOR_EXTRACTOR_DB".FIN_STK_AUTO_DN_OVR;
      A     "ONE_SECOND_PULSE";
      JNB   _046;
      L     1;
      L     "DOOR_EXTRACTOR_DB".FIN_STK_ATO_DN_DL_T;
      +I;
      T     "DOOR_EXTRACTOR_DB".FIN_STK_ATO_DN_DL_T;
_046: NOP   0;
      A     L 0.0;
      A(;
      L     "DOOR_EXTRACTOR_DB".FIN_STK_ATO_DN_DL_T;
      L     "DOOR_EXTRACTOR_DB".FIN_STK_AUTO_DN_DEL;
      >=I;
      );
      =     "DOOR_EXTRACTOR_DB".FIN_STK_AUTO_DN_OVR;
NETWORK
TITLE =
      A     "ALWAYS_ON";
      A(;
      A     "DOOR_EXTRACTOR_DB".FIN_STK_DN_CMD;
      A     "HALF_SECOND_PULSE_TRAIN";
      O     "DOOR_EXTRACTOR_DB".FIN_STK_DN_OP_CUT;
      O     "MAIN_POWER_DB".LAMP_TEST_PB;
      );
      =     "DOOR_EXTRACTOR_DB".FIN_STK_DN_IND;
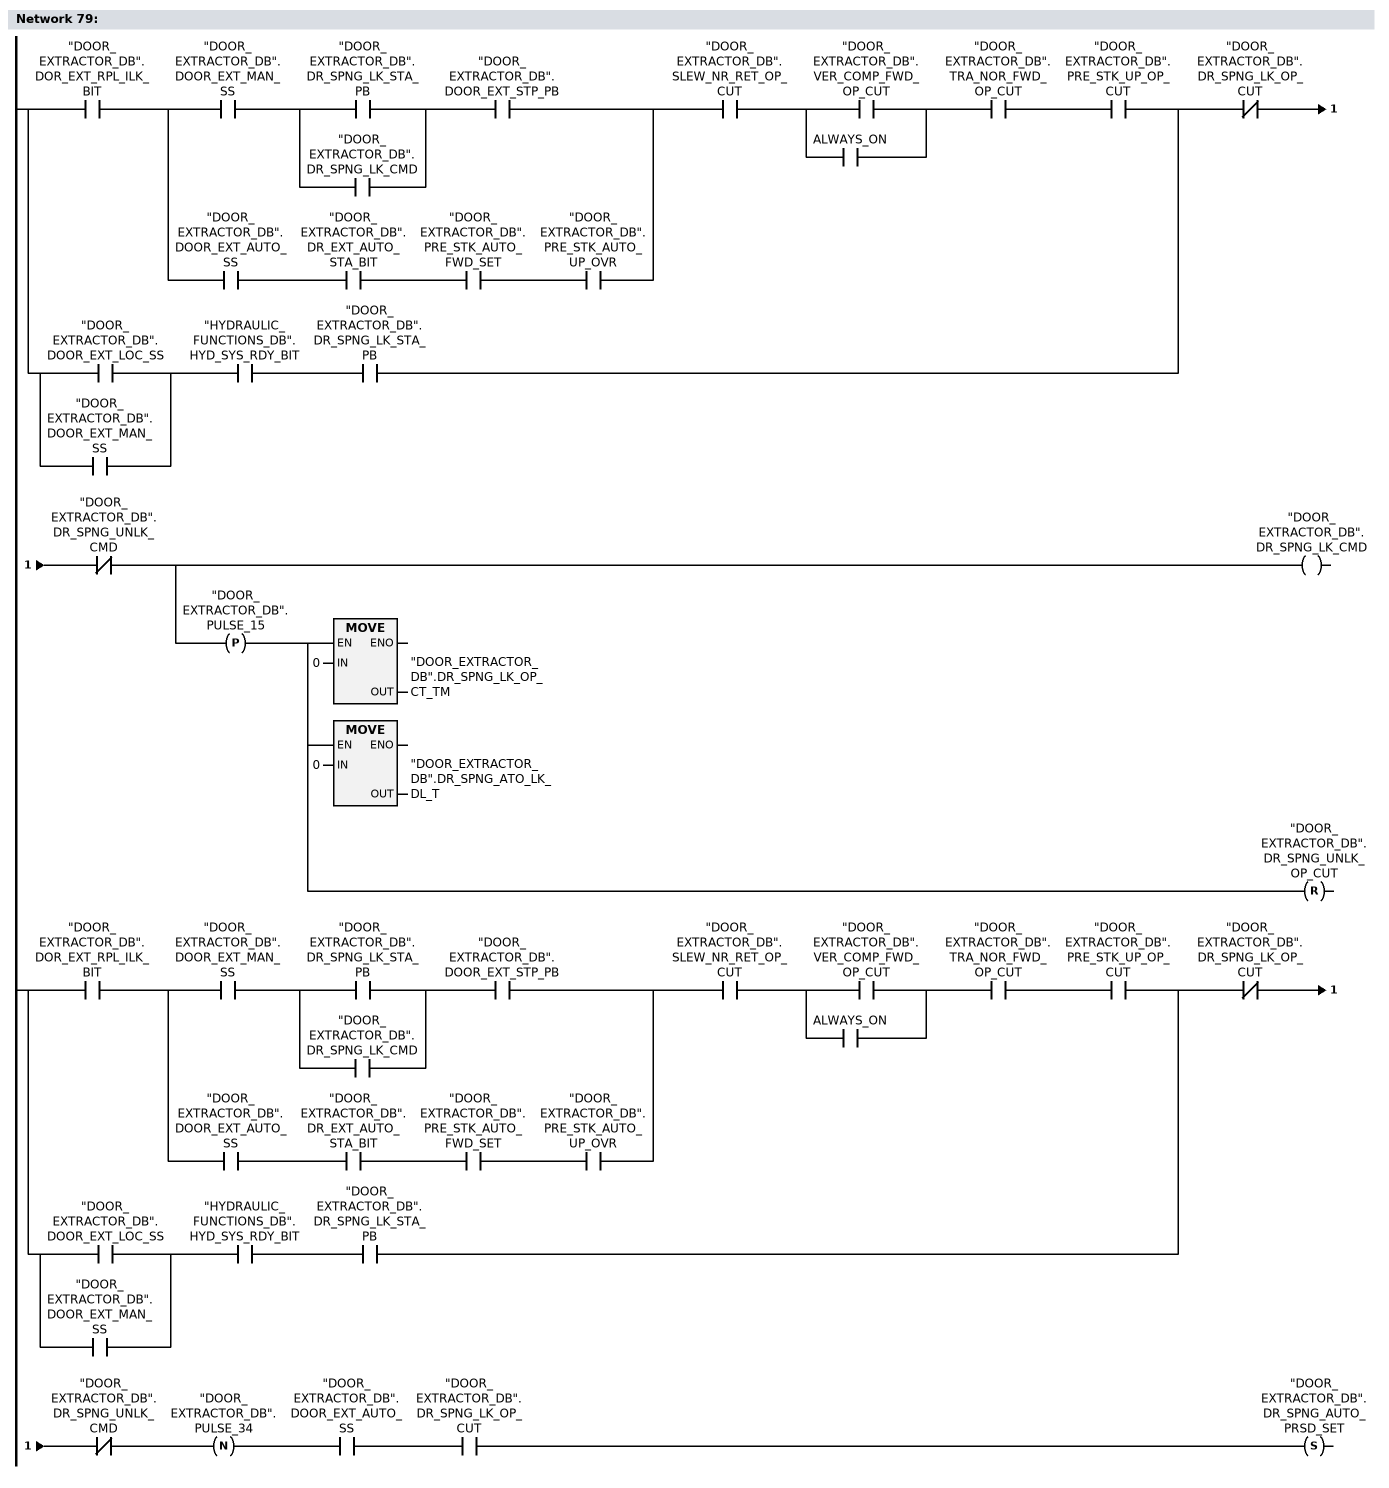
NETWORK
TITLE =
      A(;
      A     "DOOR_EXTRACTOR_DB".DOR_EXT_RPL_ILK_BIT;
      A(;
      A     "DOOR_EXTRACTOR_DB".DOOR_EXT_MAN_SS;
      A(;
      O     "DOOR_EXTRACTOR_DB".DR_SPNG_LK_STA_PB;
      O     "DOOR_EXTRACTOR_DB".DR_SPNG_LK_CMD;
      );
      A     "DOOR_EXTRACTOR_DB".DOOR_EXT_STP_PB;
      O;
      A     "DOOR_EXTRACTOR_DB".DOOR_EXT_AUTO_SS;
      A     "DOOR_EXTRACTOR_DB".DR_EXT_AUTO_STA_BIT;
      A     "DOOR_EXTRACTOR_DB".PRE_STK_AUTO_FWD_SET;
      A     "DOOR_EXTRACTOR_DB".PRE_STK_AUTO_UP_OVR;
      );
      A     "DOOR_EXTRACTOR_DB".SLEW_NR_RET_OP_CUT;
      A(;
      O     "DOOR_EXTRACTOR_DB".VER_COMP_FWD_OP_CUT;
      O     "ALWAYS_ON";
      );
      A     "DOOR_EXTRACTOR_DB".TRA_NOR_FWD_OP_CUT;
      A     "DOOR_EXTRACTOR_DB".PRE_STK_UP_OP_CUT;
      O;
      A(;
      O     "DOOR_EXTRACTOR_DB".DOOR_EXT_LOC_SS;
      O     "DOOR_EXTRACTOR_DB".DOOR_EXT_MAN_SS;
      );
      A     "HYDRAULIC_FUNCTIONS_DB".HYD_SYS_RDY_BIT;
      A     "DOOR_EXTRACTOR_DB".DR_SPNG_LK_STA_PB;
      );
      AN    "DOOR_EXTRACTOR_DB".DR_SPNG_LK_OP_CUT;
      AN    "DOOR_EXTRACTOR_DB".DR_SPNG_UNLK_CMD;
      =     L 0.0;
      A     L 0.0;
      BLD   102;
      =     "DOOR_EXTRACTOR_DB".DR_SPNG_LK_CMD;
      A(;
      A     L 0.0;
      FN    "DOOR_EXTRACTOR_DB".PULSE_34;
      );
      A     "DOOR_EXTRACTOR_DB".DOOR_EXT_AUTO_SS;
      A     "DOOR_EXTRACTOR_DB".DR_SPNG_LK_OP_CUT;
      S     "DOOR_EXTRACTOR_DB".DR_SPNG_AUTO_PRSD_SET;
      A     L 0.0;
      FP    "DOOR_EXTRACTOR_DB".PULSE_15;
      =     L 0.1;
      A     L 0.1;
      JNB   _047;
      L     0;
      T     "DOOR_EXTRACTOR_DB".DR_SPNG_LK_OP_CT_TM;
_047: NOP   0;
      A     L 0.1;
      JNB   _048;
      L     0;
      T     "DOOR_EXTRACTOR_DB".DR_SPNG_ATO_LK_DL_T;
_048: NOP   0;
      A     L 0.1;
      BLD   102;
      R     "DOOR_EXTRACTOR_DB".DR_SPNG_UNLK_OP_CUT;
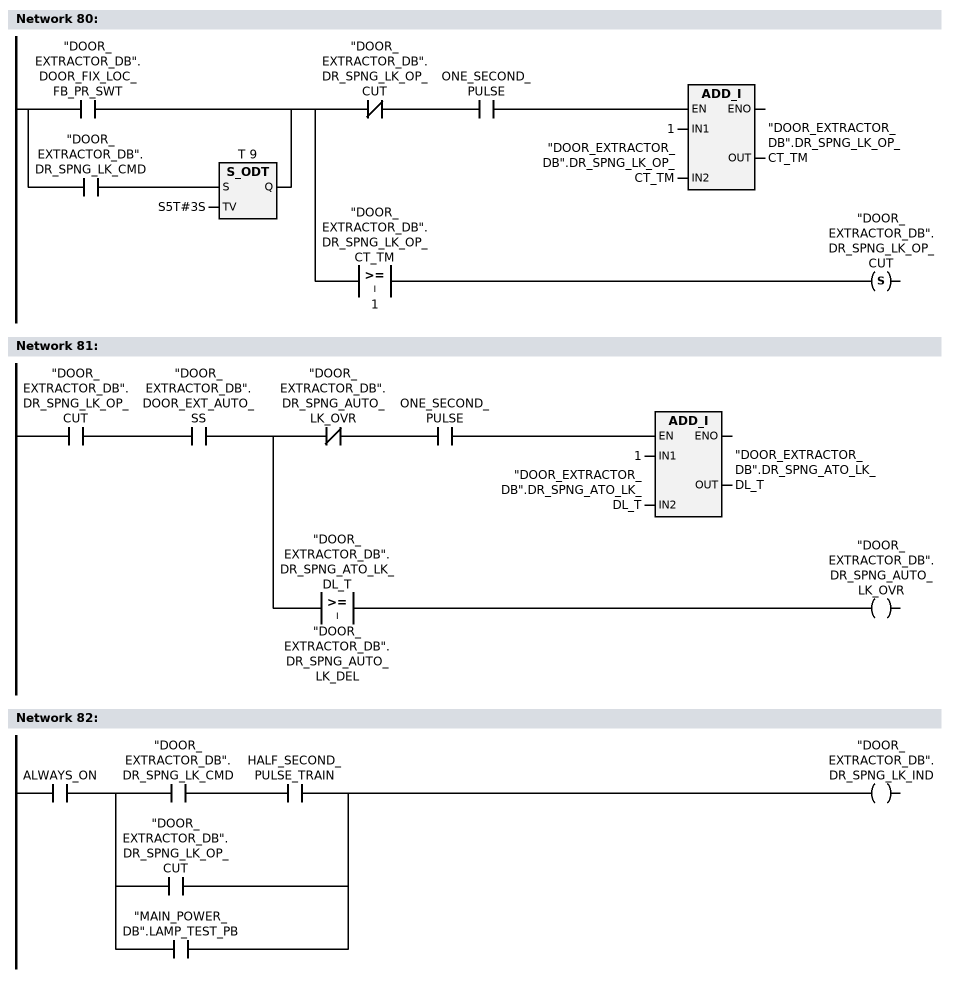
NETWORK
TITLE =
      O     "DOOR_EXTRACTOR_DB".DOOR_FIX_LOC_FB_PR_SWT;
      O(;
      A     "DOOR_EXTRACTOR_DB".DR_SPNG_LK_CMD;
      L     S5T#3S;
      SD    T 9;
      NOP   0;
      NOP   0;
      NOP   0;
      A     T 9;
      );
      =     L 0.0;
      A     L 0.0;
      AN    "DOOR_EXTRACTOR_DB".DR_SPNG_LK_OP_CUT;
      A     "ONE_SECOND_PULSE";
      JNB   _049;
      L     1;
      L     "DOOR_EXTRACTOR_DB".DR_SPNG_LK_OP_CT_TM;
      +I;
      T     "DOOR_EXTRACTOR_DB".DR_SPNG_LK_OP_CT_TM;
_049: NOP   0;
      A     L 0.0;
      A(;
      L     "DOOR_EXTRACTOR_DB".DR_SPNG_LK_OP_CT_TM;
      L     1;
      >=I;
      );
      S     "DOOR_EXTRACTOR_DB".DR_SPNG_LK_OP_CUT;
NETWORK
TITLE =
      A     "DOOR_EXTRACTOR_DB".DR_SPNG_LK_OP_CUT;
      A     "DOOR_EXTRACTOR_DB".DOOR_EXT_AUTO_SS;
      =     L 0.0;
      A     L 0.0;
      AN    "DOOR_EXTRACTOR_DB".DR_SPNG_AUTO_LK_OVR;
      A     "ONE_SECOND_PULSE";
      JNB   _04a;
      L     1;
      L     "DOOR_EXTRACTOR_DB".DR_SPNG_ATO_LK_DL_T;
      +I;
      T     "DOOR_EXTRACTOR_DB".DR_SPNG_ATO_LK_DL_T;
_04a: NOP   0;
      A     L 0.0;
      A(;
      L     "DOOR_EXTRACTOR_DB".DR_SPNG_ATO_LK_DL_T;
      L     "DOOR_EXTRACTOR_DB".DR_SPNG_AUTO_LK_DEL;
      >=I;
      );
      =     "DOOR_EXTRACTOR_DB".DR_SPNG_AUTO_LK_OVR;
NETWORK
TITLE =
      A     "ALWAYS_ON";
      A(;
      A     "DOOR_EXTRACTOR_DB".DR_SPNG_LK_CMD;
      A     "HALF_SECOND_PULSE_TRAIN";
      O     "DOOR_EXTRACTOR_DB".DR_SPNG_LK_OP_CUT;
      O     "MAIN_POWER_DB".LAMP_TEST_PB;
      );
      =     "DOOR_EXTRACTOR_DB".DR_SPNG_LK_IND;
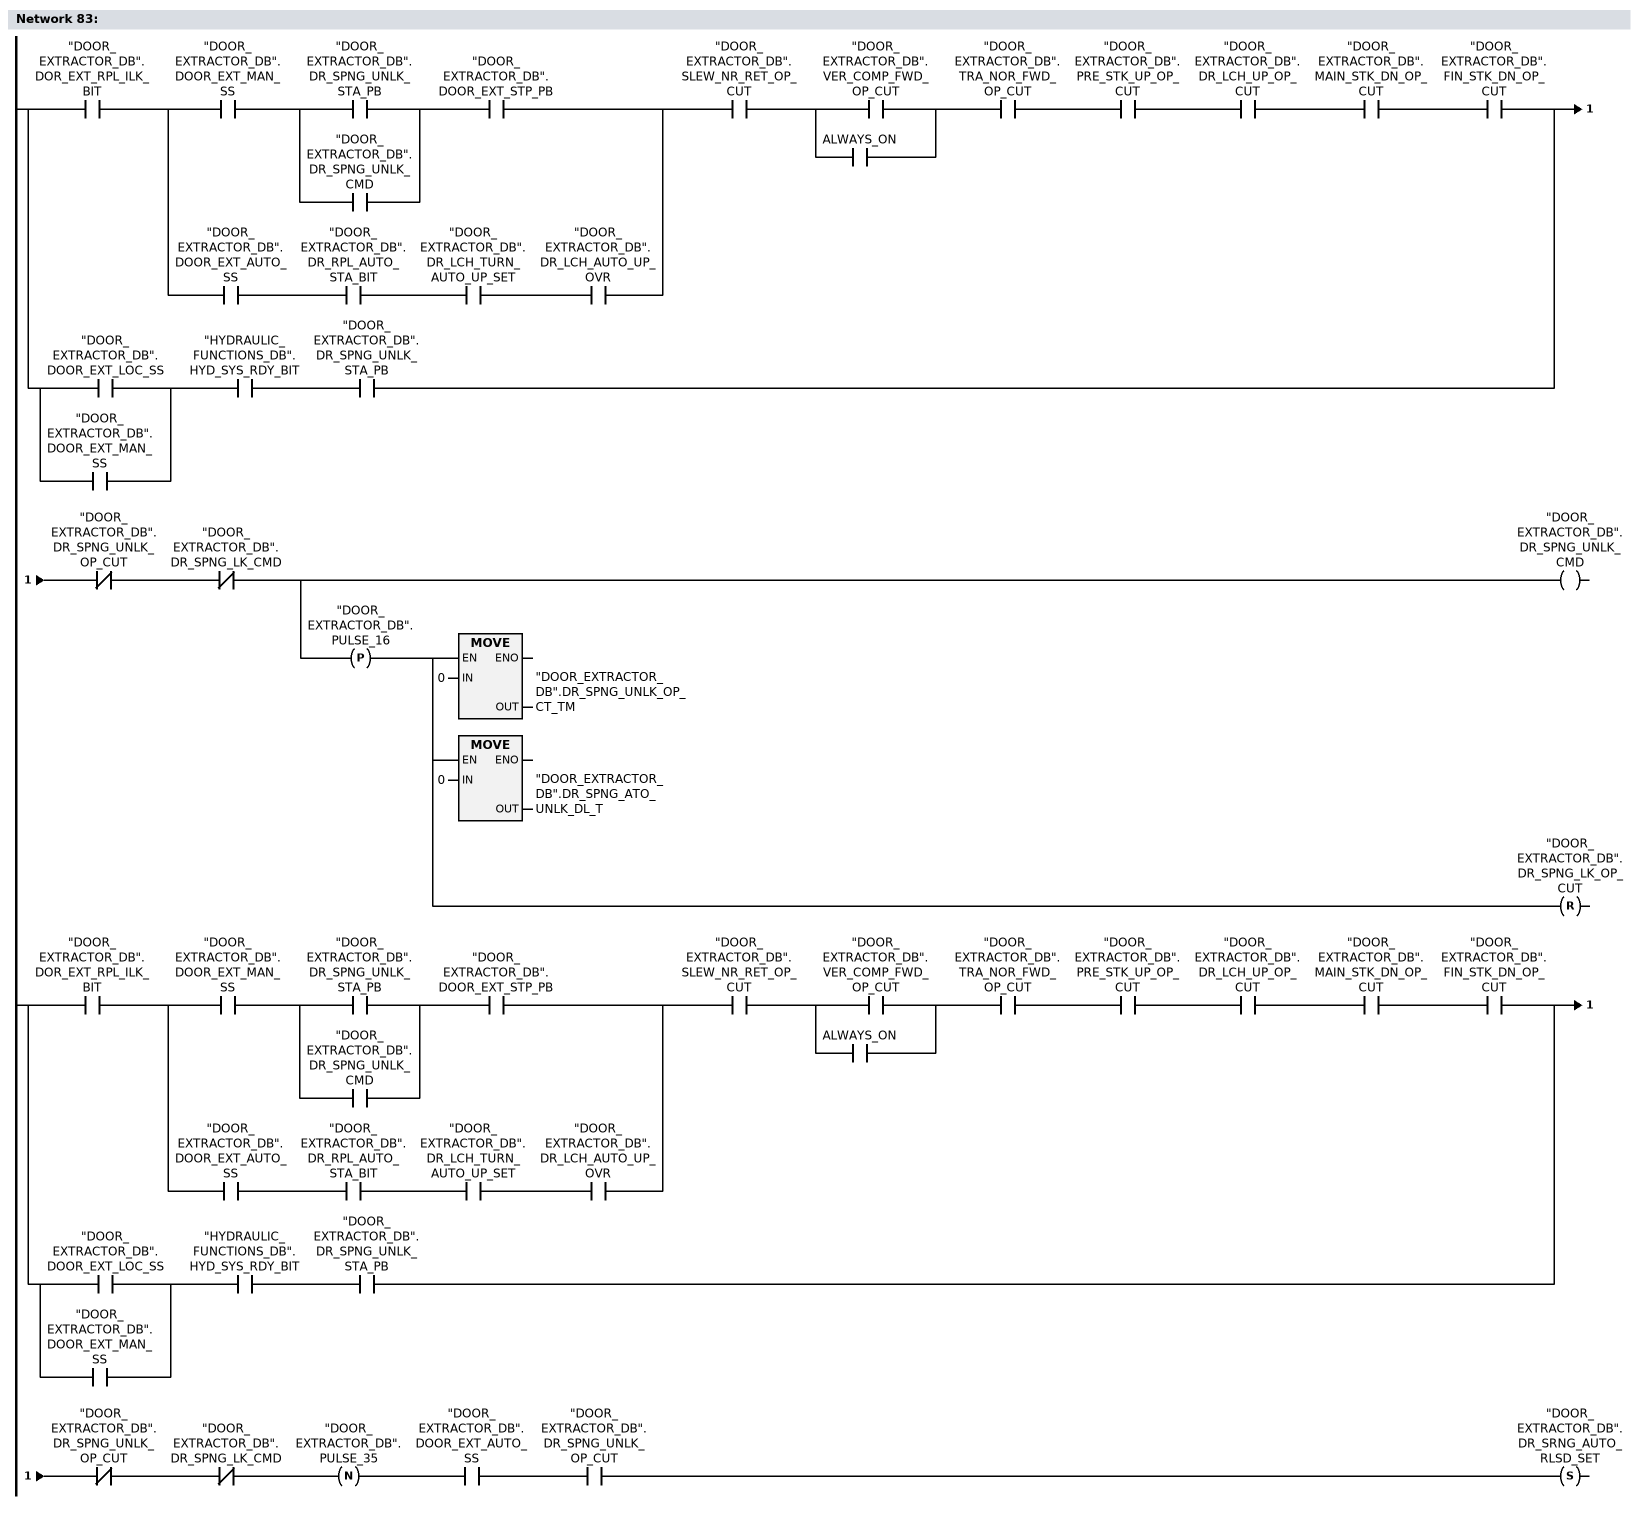
NETWORK
TITLE =
      A(;
      A     "DOOR_EXTRACTOR_DB".DOR_EXT_RPL_ILK_BIT;
      A(;
      A     "DOOR_EXTRACTOR_DB".DOOR_EXT_MAN_SS;
      A(;
      O     "DOOR_EXTRACTOR_DB".DR_SPNG_UNLK_STA_PB;
      O     "DOOR_EXTRACTOR_DB".DR_SPNG_UNLK_CMD;
      );
      A     "DOOR_EXTRACTOR_DB".DOOR_EXT_STP_PB;
      O;
      A     "DOOR_EXTRACTOR_DB".DOOR_EXT_AUTO_SS;
      A     "DOOR_EXTRACTOR_DB".DR_RPL_AUTO_STA_BIT;
      A     "DOOR_EXTRACTOR_DB".DR_LCH_TURN_AUTO_UP_SET;
      A     "DOOR_EXTRACTOR_DB".DR_LCH_AUTO_UP_OVR;
      );
      A     "DOOR_EXTRACTOR_DB".SLEW_NR_RET_OP_CUT;
      A(;
      O     "DOOR_EXTRACTOR_DB".VER_COMP_FWD_OP_CUT;
      O     "ALWAYS_ON";
      );
      A     "DOOR_EXTRACTOR_DB".TRA_NOR_FWD_OP_CUT;
      A     "DOOR_EXTRACTOR_DB".PRE_STK_UP_OP_CUT;
      A     "DOOR_EXTRACTOR_DB".DR_LCH_UP_OP_CUT;
      A     "DOOR_EXTRACTOR_DB".MAIN_STK_DN_OP_CUT;
      A     "DOOR_EXTRACTOR_DB".FIN_STK_DN_OP_CUT;
      O;
      A(;
      O     "DOOR_EXTRACTOR_DB".DOOR_EXT_LOC_SS;
      O     "DOOR_EXTRACTOR_DB".DOOR_EXT_MAN_SS;
      );
      A     "HYDRAULIC_FUNCTIONS_DB".HYD_SYS_RDY_BIT;
      A     "DOOR_EXTRACTOR_DB".DR_SPNG_UNLK_STA_PB;
      );
      AN    "DOOR_EXTRACTOR_DB".DR_SPNG_UNLK_OP_CUT;
      AN    "DOOR_EXTRACTOR_DB".DR_SPNG_LK_CMD;
      =     L 0.0;
      A     L 0.0;
      BLD   102;
      =     "DOOR_EXTRACTOR_DB".DR_SPNG_UNLK_CMD;
      A(;
      A     L 0.0;
      FN    "DOOR_EXTRACTOR_DB".PULSE_35;
      );
      A     "DOOR_EXTRACTOR_DB".DOOR_EXT_AUTO_SS;
      A     "DOOR_EXTRACTOR_DB".DR_SPNG_UNLK_OP_CUT;
      S     "DOOR_EXTRACTOR_DB".DR_SRNG_AUTO_RLSD_SET;
      A     L 0.0;
      FP    "DOOR_EXTRACTOR_DB".PULSE_16;
      =     L 0.1;
      A     L 0.1;
      JNB   _04b;
      L     0;
      T     "DOOR_EXTRACTOR_DB".DR_SPNG_UNLK_OP_CT_TM;
_04b: NOP   0;
      A     L 0.1;
      JNB   _04c;
      L     0;
      T     "DOOR_EXTRACTOR_DB".DR_SPNG_ATO_UNLK_DL_T;
_04c: NOP   0;
      A     L 0.1;
      BLD   102;
      R     "DOOR_EXTRACTOR_DB".DR_SPNG_LK_OP_CUT;
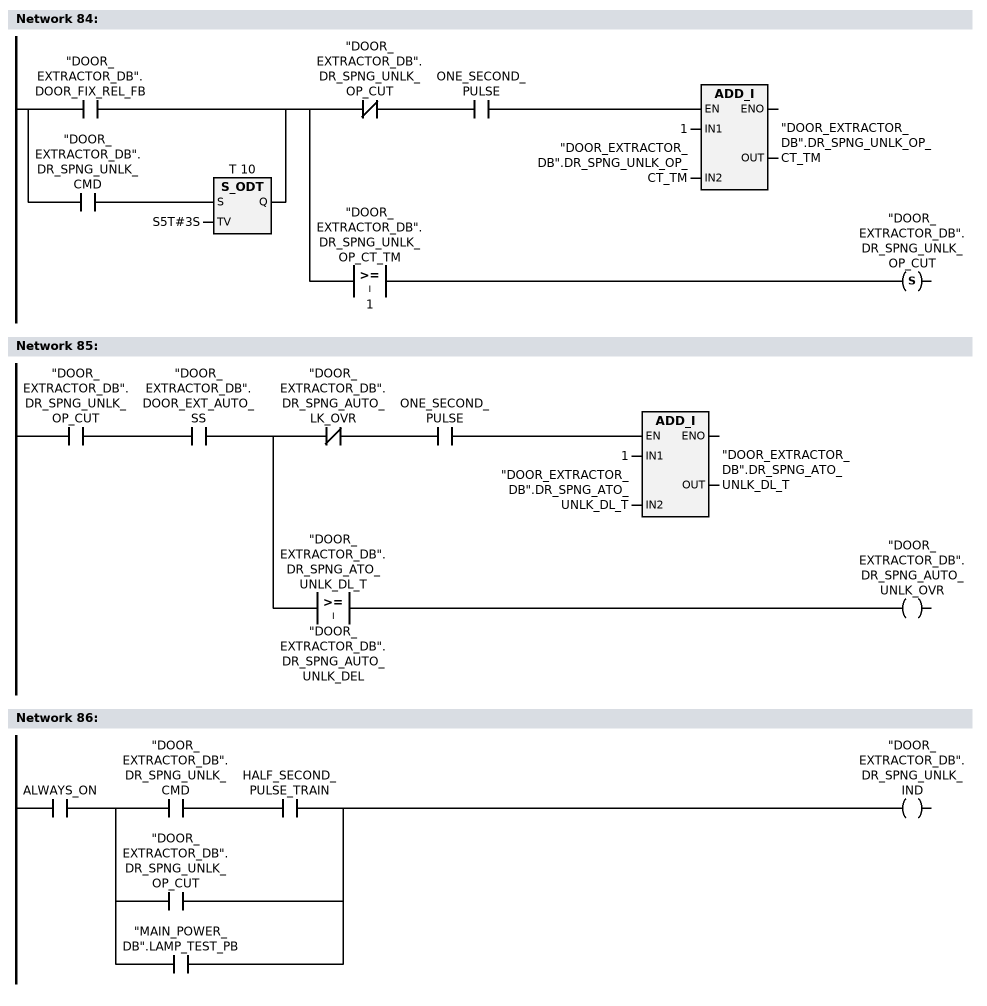
NETWORK
TITLE =
      O     "DOOR_EXTRACTOR_DB".DOOR_FIX_REL_FB;
      O(;
      A     "DOOR_EXTRACTOR_DB".DR_SPNG_UNLK_CMD;
      L     S5T#3S;
      SD    T 10;
      NOP   0;
      NOP   0;
      NOP   0;
      A     T 10;
      );
      =     L 0.0;
      A     L 0.0;
      AN    "DOOR_EXTRACTOR_DB".DR_SPNG_UNLK_OP_CUT;
      A     "ONE_SECOND_PULSE";
      JNB   _04d;
      L     1;
      L     "DOOR_EXTRACTOR_DB".DR_SPNG_UNLK_OP_CT_TM;
      +I;
      T     "DOOR_EXTRACTOR_DB".DR_SPNG_UNLK_OP_CT_TM;
_04d: NOP   0;
      A     L 0.0;
      A(;
      L     "DOOR_EXTRACTOR_DB".DR_SPNG_UNLK_OP_CT_TM;
      L     1;
      >=I;
      );
      S     "DOOR_EXTRACTOR_DB".DR_SPNG_UNLK_OP_CUT;
NETWORK
TITLE =
      A     "DOOR_EXTRACTOR_DB".DR_SPNG_UNLK_OP_CUT;
      A     "DOOR_EXTRACTOR_DB".DOOR_EXT_AUTO_SS;
      =     L 0.0;
      A     L 0.0;
      AN    "DOOR_EXTRACTOR_DB".DR_SPNG_AUTO_LK_OVR;
      A     "ONE_SECOND_PULSE";
      JNB   _04e;
      L     1;
      L     "DOOR_EXTRACTOR_DB".DR_SPNG_ATO_UNLK_DL_T;
      +I;
      T     "DOOR_EXTRACTOR_DB".DR_SPNG_ATO_UNLK_DL_T;
_04e: NOP   0;
      A     L 0.0;
      A(;
      L     "DOOR_EXTRACTOR_DB".DR_SPNG_ATO_UNLK_DL_T;
      L     "DOOR_EXTRACTOR_DB".DR_SPNG_AUTO_UNLK_DEL;
      >=I;
      );
      =     "DOOR_EXTRACTOR_DB".DR_SPNG_AUTO_UNLK_OVR;
NETWORK
TITLE =
      A     "ALWAYS_ON";
      A(;
      A     "DOOR_EXTRACTOR_DB".DR_SPNG_UNLK_CMD;
      A     "HALF_SECOND_PULSE_TRAIN";
      O     "DOOR_EXTRACTOR_DB".DR_SPNG_UNLK_OP_CUT;
      O     "MAIN_POWER_DB".LAMP_TEST_PB;
      );
      =     "DOOR_EXTRACTOR_DB".DR_SPNG_UNLK_IND;
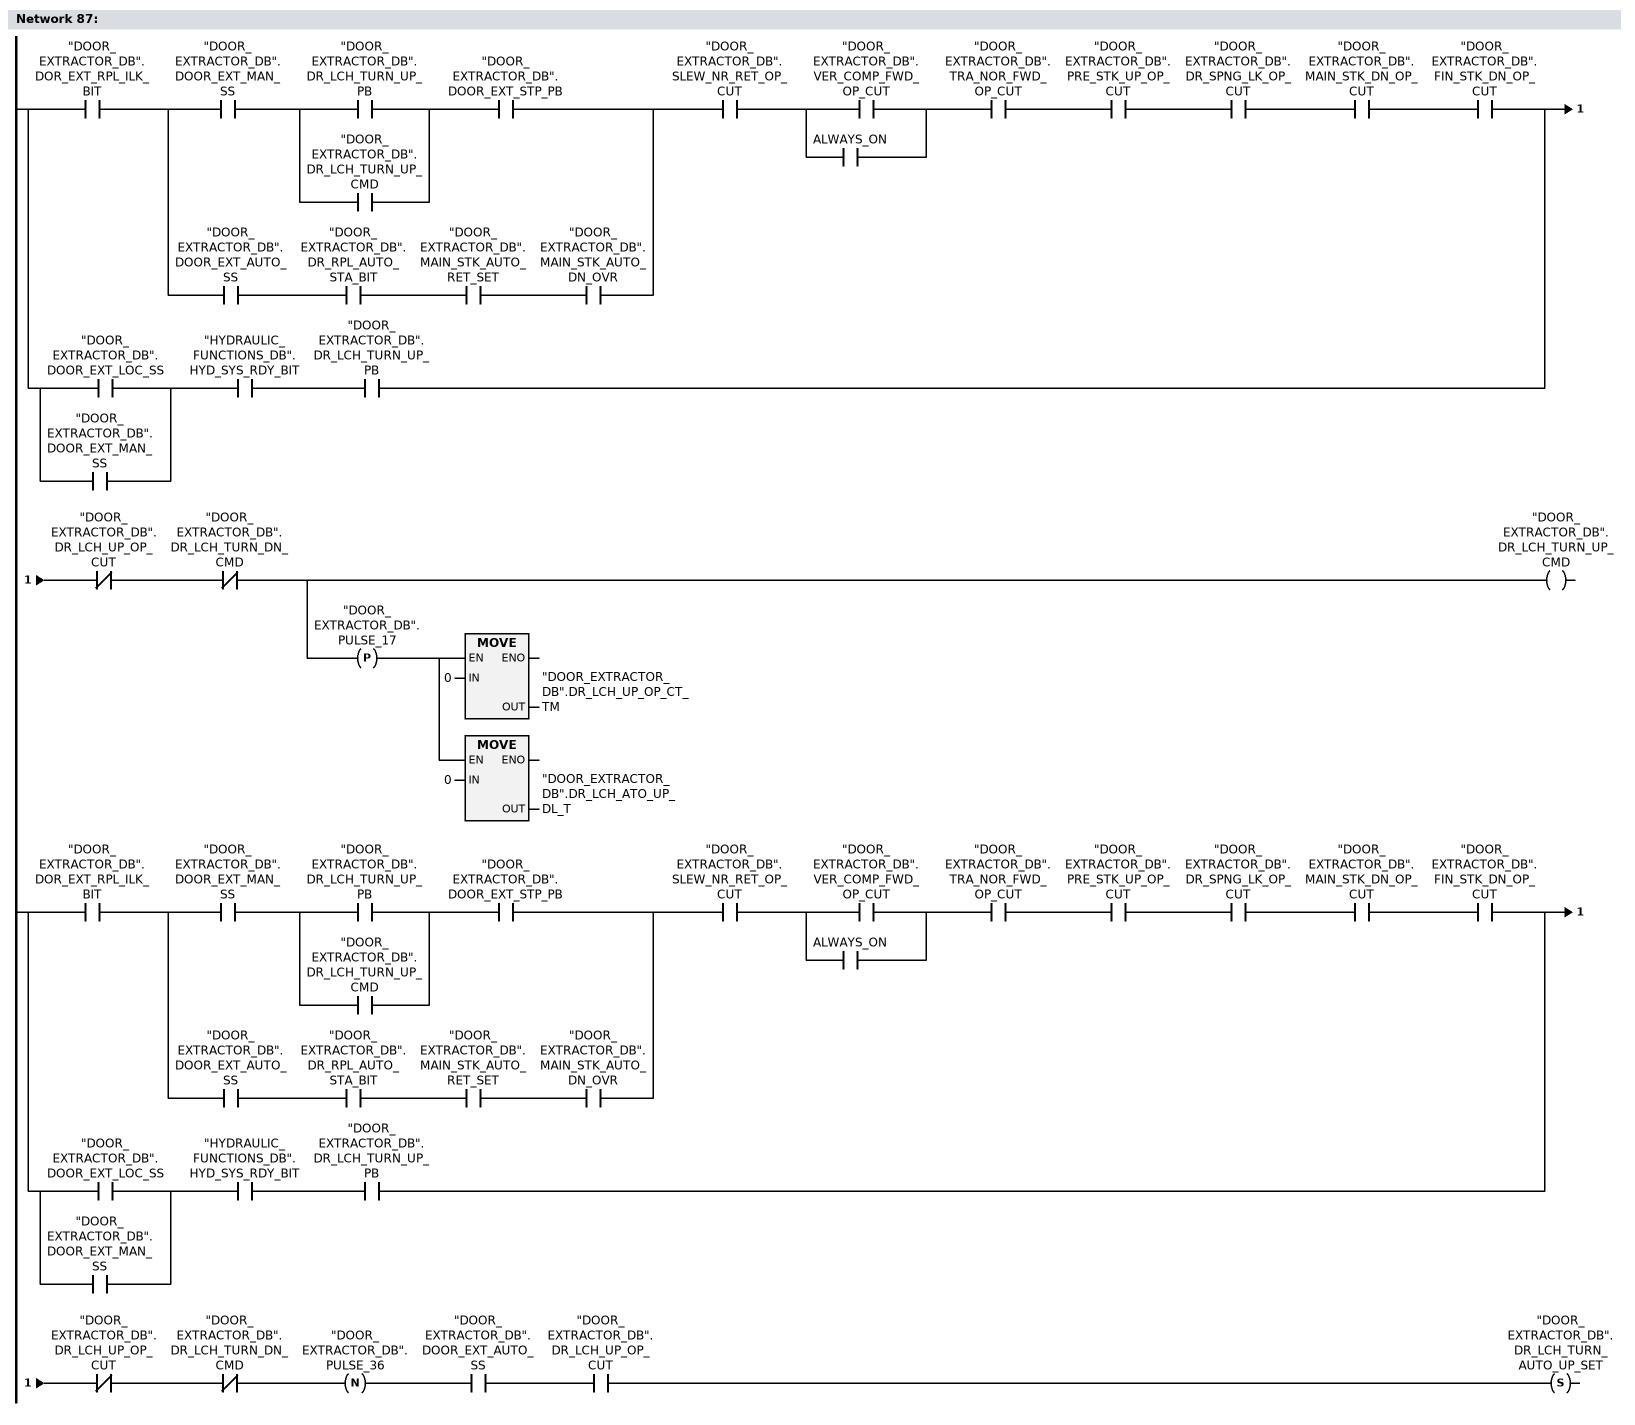
NETWORK
TITLE =
      A(;
      A     "DOOR_EXTRACTOR_DB".DOR_EXT_RPL_ILK_BIT;
      A(;
      A     "DOOR_EXTRACTOR_DB".DOOR_EXT_MAN_SS;
      A(;
      O     "DOOR_EXTRACTOR_DB".DR_LCH_TURN_UP_PB;
      O     "DOOR_EXTRACTOR_DB".DR_LCH_TURN_UP_CMD;
      );
      A     "DOOR_EXTRACTOR_DB".DOOR_EXT_STP_PB;
      O;
      A     "DOOR_EXTRACTOR_DB".DOOR_EXT_AUTO_SS;
      A     "DOOR_EXTRACTOR_DB".DR_RPL_AUTO_STA_BIT;
      A     "DOOR_EXTRACTOR_DB".MAIN_STK_AUTO_RET_SET;
      A     "DOOR_EXTRACTOR_DB".MAIN_STK_AUTO_DN_OVR;
      );
      A     "DOOR_EXTRACTOR_DB".SLEW_NR_RET_OP_CUT;
      A(;
      O     "DOOR_EXTRACTOR_DB".VER_COMP_FWD_OP_CUT;
      O     "ALWAYS_ON";
      );
      A     "DOOR_EXTRACTOR_DB".TRA_NOR_FWD_OP_CUT;
      A     "DOOR_EXTRACTOR_DB".PRE_STK_UP_OP_CUT;
      A     "DOOR_EXTRACTOR_DB".DR_SPNG_LK_OP_CUT;
      A     "DOOR_EXTRACTOR_DB".MAIN_STK_DN_OP_CUT;
      A     "DOOR_EXTRACTOR_DB".FIN_STK_DN_OP_CUT;
      O;
      A(;
      O     "DOOR_EXTRACTOR_DB".DOOR_EXT_LOC_SS;
      O     "DOOR_EXTRACTOR_DB".DOOR_EXT_MAN_SS;
      );
      A     "HYDRAULIC_FUNCTIONS_DB".HYD_SYS_RDY_BIT;
      A     "DOOR_EXTRACTOR_DB".DR_LCH_TURN_UP_PB;
      );
      AN    "DOOR_EXTRACTOR_DB".DR_LCH_UP_OP_CUT;
      AN    "DOOR_EXTRACTOR_DB".DR_LCH_TURN_DN_CMD;
      =     L 0.0;
      A     L 0.0;
      BLD   102;
      =     "DOOR_EXTRACTOR_DB".DR_LCH_TURN_UP_CMD;
      A(;
      A     L 0.0;
      FN    "DOOR_EXTRACTOR_DB".PULSE_36;
      );
      A     "DOOR_EXTRACTOR_DB".DOOR_EXT_AUTO_SS;
      A     "DOOR_EXTRACTOR_DB".DR_LCH_UP_OP_CUT;
      S     "DOOR_EXTRACTOR_DB".DR_LCH_TURN_AUTO_UP_SET;
      A     L 0.0;
      FP    "DOOR_EXTRACTOR_DB".PULSE_17;
      =     L 0.1;
      A     L 0.1;
      JNB   _04f;
      L     0;
      T     "DOOR_EXTRACTOR_DB".DR_LCH_UP_OP_CT_TM;
_04f: NOP   0;
      A     L 0.1;
      JNB   _050;
      L     0;
      T     "DOOR_EXTRACTOR_DB".DR_LCH_ATO_UP_DL_T;
_050: NOP   0;
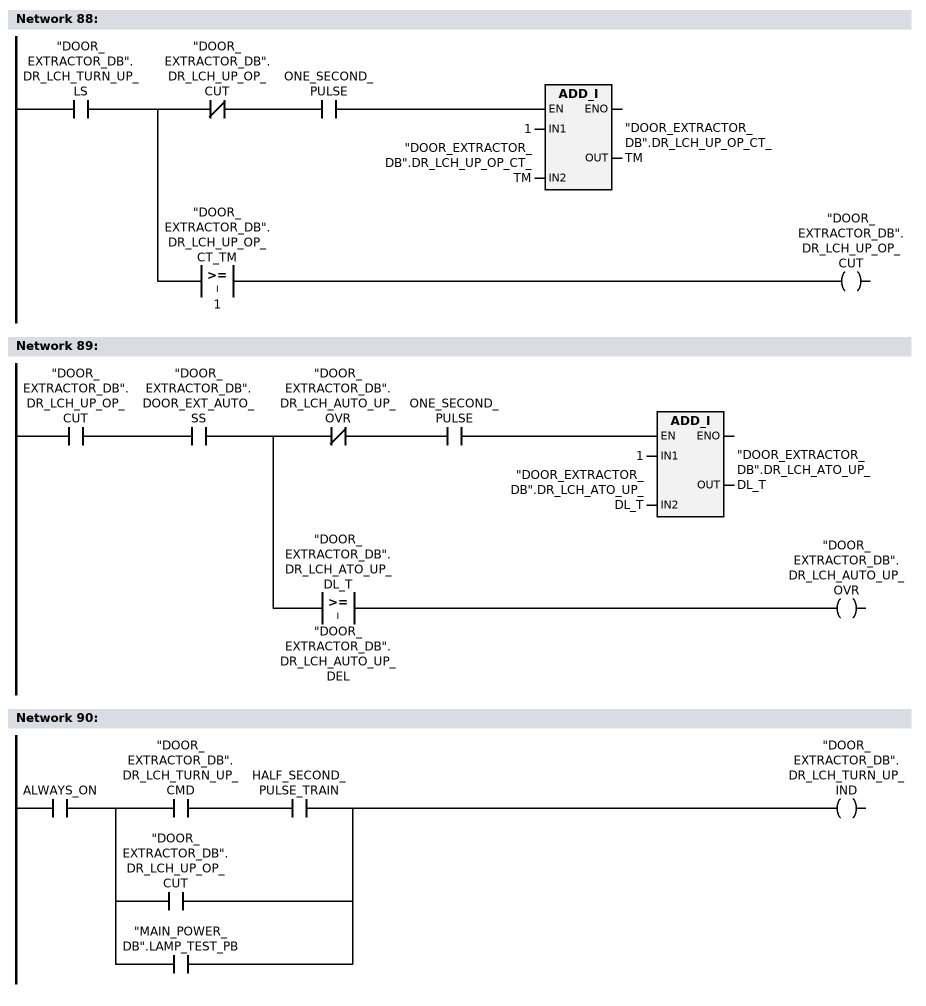
NETWORK
TITLE =
      A     "DOOR_EXTRACTOR_DB".DR_LCH_TURN_UP_LS;
      =     L 0.0;
      A     L 0.0;
      AN    "DOOR_EXTRACTOR_DB".DR_LCH_UP_OP_CUT;
      A     "ONE_SECOND_PULSE";
      JNB   _051;
      L     1;
      L     "DOOR_EXTRACTOR_DB".DR_LCH_UP_OP_CT_TM;
      +I;
      T     "DOOR_EXTRACTOR_DB".DR_LCH_UP_OP_CT_TM;
_051: NOP   0;
      A     L 0.0;
      A(;
      L     "DOOR_EXTRACTOR_DB".DR_LCH_UP_OP_CT_TM;
      L     1;
      >=I;
      );
      =     "DOOR_EXTRACTOR_DB".DR_LCH_UP_OP_CUT;
NETWORK
TITLE =
      A     "DOOR_EXTRACTOR_DB".DR_LCH_UP_OP_CUT;
      A     "DOOR_EXTRACTOR_DB".DOOR_EXT_AUTO_SS;
      =     L 0.0;
      A     L 0.0;
      AN    "DOOR_EXTRACTOR_DB".DR_LCH_AUTO_UP_OVR;
      A     "ONE_SECOND_PULSE";
      JNB   _052;
      L     1;
      L     "DOOR_EXTRACTOR_DB".DR_LCH_ATO_UP_DL_T;
      +I;
      T     "DOOR_EXTRACTOR_DB".DR_LCH_ATO_UP_DL_T;
_052: NOP   0;
      A     L 0.0;
      A(;
      L     "DOOR_EXTRACTOR_DB".DR_LCH_ATO_UP_DL_T;
      L     "DOOR_EXTRACTOR_DB".DR_LCH_AUTO_UP_DEL;
      >=I;
      );
      =     "DOOR_EXTRACTOR_DB".DR_LCH_AUTO_UP_OVR;
NETWORK
TITLE =
      A     "ALWAYS_ON";
      A(;
      A     "DOOR_EXTRACTOR_DB".DR_LCH_TURN_UP_CMD;
      A     "HALF_SECOND_PULSE_TRAIN";
      O     "DOOR_EXTRACTOR_DB".DR_LCH_UP_OP_CUT;
      O     "MAIN_POWER_DB".LAMP_TEST_PB;
      );
      =     "DOOR_EXTRACTOR_DB".DR_LCH_TURN_UP_IND;
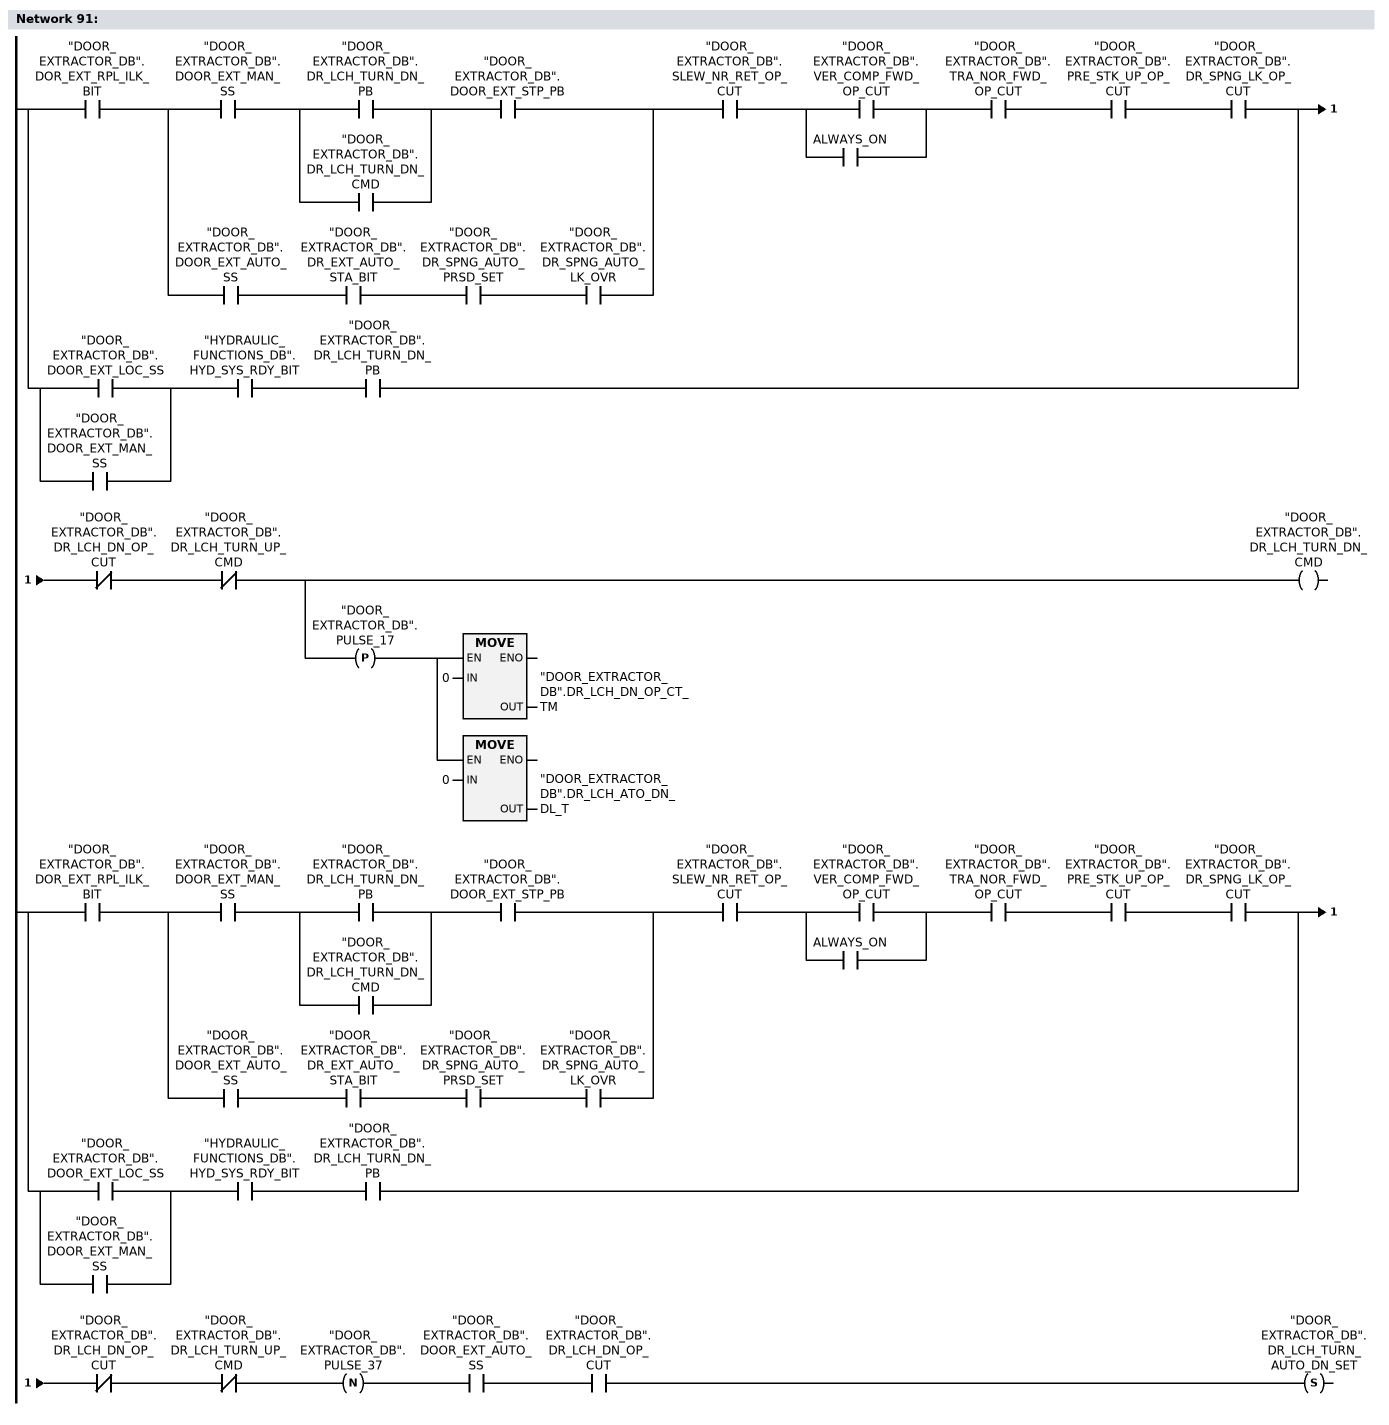
NETWORK
TITLE =
      A(;
      A     "DOOR_EXTRACTOR_DB".DOR_EXT_RPL_ILK_BIT;
      A(;
      A     "DOOR_EXTRACTOR_DB".DOOR_EXT_MAN_SS;
      A(;
      O     "DOOR_EXTRACTOR_DB".DR_LCH_TURN_DN_PB;
      O     "DOOR_EXTRACTOR_DB".DR_LCH_TURN_DN_CMD;
      );
      A     "DOOR_EXTRACTOR_DB".DOOR_EXT_STP_PB;
      O;
      A     "DOOR_EXTRACTOR_DB".DOOR_EXT_AUTO_SS;
      A     "DOOR_EXTRACTOR_DB".DR_EXT_AUTO_STA_BIT;
      A     "DOOR_EXTRACTOR_DB".DR_SPNG_AUTO_PRSD_SET;
      A     "DOOR_EXTRACTOR_DB".DR_SPNG_AUTO_LK_OVR;
      );
      A     "DOOR_EXTRACTOR_DB".SLEW_NR_RET_OP_CUT;
      A(;
      O     "DOOR_EXTRACTOR_DB".VER_COMP_FWD_OP_CUT;
      O     "ALWAYS_ON";
      );
      A     "DOOR_EXTRACTOR_DB".TRA_NOR_FWD_OP_CUT;
      A     "DOOR_EXTRACTOR_DB".PRE_STK_UP_OP_CUT;
      A     "DOOR_EXTRACTOR_DB".DR_SPNG_LK_OP_CUT;
      O;
      A(;
      O     "DOOR_EXTRACTOR_DB".DOOR_EXT_LOC_SS;
      O     "DOOR_EXTRACTOR_DB".DOOR_EXT_MAN_SS;
      );
      A     "HYDRAULIC_FUNCTIONS_DB".HYD_SYS_RDY_BIT;
      A     "DOOR_EXTRACTOR_DB".DR_LCH_TURN_DN_PB;
      );
      AN    "DOOR_EXTRACTOR_DB".DR_LCH_DN_OP_CUT;
      AN    "DOOR_EXTRACTOR_DB".DR_LCH_TURN_UP_CMD;
      =     L 0.0;
      A     L 0.0;
      BLD   102;
      =     "DOOR_EXTRACTOR_DB".DR_LCH_TURN_DN_CMD;
      A(;
      A     L 0.0;
      FN    "DOOR_EXTRACTOR_DB".PULSE_37;
      );
      A     "DOOR_EXTRACTOR_DB".DOOR_EXT_AUTO_SS;
      A     "DOOR_EXTRACTOR_DB".DR_LCH_DN_OP_CUT;
      S     "DOOR_EXTRACTOR_DB".DR_LCH_TURN_AUTO_DN_SET;
      A     L 0.0;
      FP    "DOOR_EXTRACTOR_DB".PULSE_17;
      =     L 0.1;
      A     L 0.1;
      JNB   _053;
      L     0;
      T     "DOOR_EXTRACTOR_DB".DR_LCH_DN_OP_CT_TM;
_053: NOP   0;
      A     L 0.1;
      JNB   _054;
      L     0;
      T     "DOOR_EXTRACTOR_DB".DR_LCH_ATO_DN_DL_T;
_054: NOP   0;
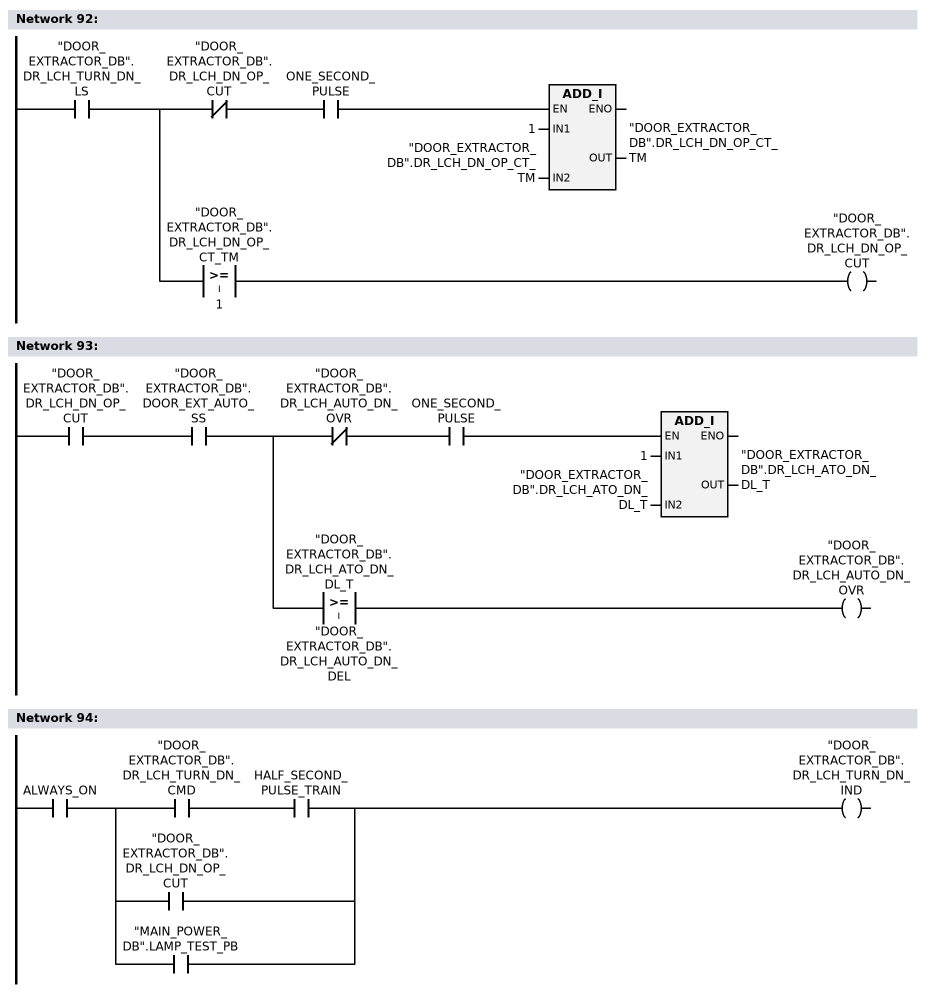
NETWORK
TITLE =
      A     "DOOR_EXTRACTOR_DB".DR_LCH_TURN_DN_LS;
      =     L 0.0;
      A     L 0.0;
      AN    "DOOR_EXTRACTOR_DB".DR_LCH_DN_OP_CUT;
      A     "ONE_SECOND_PULSE";
      JNB   _055;
      L     1;
      L     "DOOR_EXTRACTOR_DB".DR_LCH_DN_OP_CT_TM;
      +I;
      T     "DOOR_EXTRACTOR_DB".DR_LCH_DN_OP_CT_TM;
_055: NOP   0;
      A     L 0.0;
      A(;
      L     "DOOR_EXTRACTOR_DB".DR_LCH_DN_OP_CT_TM;
      L     1;
      >=I;
      );
      =     "DOOR_EXTRACTOR_DB".DR_LCH_DN_OP_CUT;
NETWORK
TITLE =
      A     "DOOR_EXTRACTOR_DB".DR_LCH_DN_OP_CUT;
      A     "DOOR_EXTRACTOR_DB".DOOR_EXT_AUTO_SS;
      =     L 0.0;
      A     L 0.0;
      AN    "DOOR_EXTRACTOR_DB".DR_LCH_AUTO_DN_OVR;
      A     "ONE_SECOND_PULSE";
      JNB   _056;
      L     1;
      L     "DOOR_EXTRACTOR_DB".DR_LCH_ATO_DN_DL_T;
      +I;
      T     "DOOR_EXTRACTOR_DB".DR_LCH_ATO_DN_DL_T;
_056: NOP   0;
      A     L 0.0;
      A(;
      L     "DOOR_EXTRACTOR_DB".DR_LCH_ATO_DN_DL_T;
      L     "DOOR_EXTRACTOR_DB".DR_LCH_AUTO_DN_DEL;
      >=I;
      );
      =     "DOOR_EXTRACTOR_DB".DR_LCH_AUTO_DN_OVR;
NETWORK
TITLE =
      A     "ALWAYS_ON";
      A(;
      A     "DOOR_EXTRACTOR_DB".DR_LCH_TURN_DN_CMD;
      A     "HALF_SECOND_PULSE_TRAIN";
      O     "DOOR_EXTRACTOR_DB".DR_LCH_DN_OP_CUT;
      O     "MAIN_POWER_DB".LAMP_TEST_PB;
      );
      =     "DOOR_EXTRACTOR_DB".DR_LCH_TURN_DN_IND;
END_FUNCTION

FUNCTION "SERVICE_PLATFORM" : VOID	// FC 9
AUTHOR : Kamillas
VERSION : 0.1
BEGIN
// (block stored without names or comments; labels and parameter names are numbered)
